// ---- DUTs/ST_COM_SpdCntrl_IMD.TcDUT
TYPE ST_COM_SpdCntrl_IMD :
STRUCT
	StartFormingA		: BOOL;	//Speedcontrol needs the IMD to start froming for A side	
	StartFormingB		: BOOL;	//Speedcontrol needs the IMD to start froming for B side	
	StopForming			: BOOL;					// Speedcontrol needs the IMD to stop forming 
	BlowOffPulseA		: ARRAY[1..4] OF BOOL;	// Blowoff pulses for A side
	BlowOffPulseB		: ARRAY[1..4] OF BOOL;	// Blowoff pulses for B side
	ErrSlotANotFree		: BOOL;					// Current slot for gantry A blow off was not free
	ErrSlotBNotFree		: BOOL;					// Current slot for gantry B blow off was not free
	Modulo				: LREAL;				// Actual modulo position of the belt  
	SpeedInKo			: LREAL;				//Actual Speed that speedcontrol is dictating to the IMD
	PocketA_Blocked		: BOOL;					//Pocket is occupied and gantry is not allowed to blow off
	PocketB_Blocked		: BOOL;					//Pocket is occupied and gantry is not allowed to blow off
	ProdParameters		: St_BlowOffProdPar;	// Needs to be changed to correct format
END_STRUCT
END_TYPE

// ---- DUTs/ST_Record.TcDUT
TYPE ST_Record :
	STRUCT
		nID			: LINT;
		dtTimestamp : DATE_AND_TIME;
		sName		: STRING;
		nSensor1	: LREAL;
	END_STRUCT
END_TYPE

// ---- DUTs/ST_SysPar.TcDUT
TYPE ST_SysPar :
STRUCT
	InMoldDrying					: ST_IMDSysPar;
	ProductHandling					: ST_ProductHandlingSysPar;
END_STRUCT
END_TYPE

// ---- POUs/InMoldDrying/BottomMold/ST_BottomMoldErrors.TcDUT
TYPE ST_BottomMoldErrors :
STRUCT
	VacuumSection						: ARRAY [1..GVL.MaxNrOfVacSectTakeOutUnit] OF BOOL;
	HorizontalCilinder					: ST_CilinderErrors;
	VerticalCilinder					: ST_CilinderErrors;

	Hydraulic							: ST_HydraulicErrors;
	HeatingZone 						: ARRAY [1..6] OF ST_HeatingZoneErrors;
	
	HorizontalAxis						: ST_NcAxis_Errors;
END_STRUCT
END_TYPE

// ---- POUs/InMoldDrying/BottomMold/ST_BottomMoldMachPar.TcDUT
TYPE ST_BottomMoldMachPar :
STRUCT
	EnableNewTakeOut						: BOOL;
	PositionInStop							: REAL;
	//PositionInSlow						: REAL;
	PositionOutStop							: REAL;
	PhysicalOffsetPos						: REAL;
	
	StartVacAtTrPosOffset					: REAL;	// Start vacuum position at postion x of transfer (ofset)			
	StopVacAtBmPosOffset					: REAL; // Stop vacuum at a certain bottommold pos (this is the ofset from the end)
	
	HorizontalCilinder						: ST_CilinderParameters;
	VerticalCilinder						: ST_CilinderParameters;
	
	//BottomMoldVacuumDelay					: TIME := T#22S;
	BottomMoldVacuumClosed					: TIME;
	ClosedVacEnabled						: BOOL;	

	
	VerticalCilinderUpDelay					: TIME := T#1250MS;
	VerticalCilinderTakeOutTime				: TIME := T#1250MS;
	
	
	AxisVelocityManual						: LREAL;
	AxisVelocityInit						: LREAL;
	AxisVelocityAuto						: LREAL;
	AxisPositionRest						: LREAL;
	AxisPositionHome						: LREAL;(* Used when motor is Replaced, write this value as "position bias" in system manager NC-Axis *)

	
	
	//PIDTempZone 							: ARRAY [1..6] OF ST_PIDSettings;
	HeatingZone								: ARRAY [1..6] OF ST_HeatingZone;
	VacuumSection							: ARRAY [1..6] OF FB_MonoValveNoFdbck;
	EnableVacuumSection						: ARRAY [1..6] OF BOOL;	
	
	KickOffCounter							: DINT; // Counts the number of times the bottommold moved in or out.
	GreasingVelocity						: LREAL;
	GreasingPosition						: LREAL;
	
END_STRUCT
END_TYPE

// ---- POUs/InMoldDrying/BottomMold/ST_BottomMoldProdPar.TcDUT
TYPE ST_BottomMoldProdPar :
STRUCT
	par1: REAL;
	
	
END_STRUCT
END_TYPE

// ---- POUs/InMoldDrying/BottomMold/ST_BottomMoldSysPar.TcDUT
TYPE ST_BottomMoldSysPar :
STRUCT
	BottomMoldAxis				: ST_NcAxis_SysPar;
END_STRUCT
END_TYPE

// ---- POUs/InMoldDrying/HydrolicsMain/ST_HydraulicsMainErrors.TcDUT
TYPE ST_HydraulicsMainErrors :
STRUCT
	// Alarms
	OilTemperatureTooHigh				: BOOL;
	OilLevelTooLow						: BOOL;
	Filter100Dirty						: BOOL;
	AuxFilter100Dirty					: BOOL;
	
	// Warnings
	Filter75Dirty						: BOOL;
	AuxFilter75Dirty					: BOOL;
	
	CoolingFanCabinet					: BOOL;
	Hydraulics24VError					: BOOL;
	
	
	// Alarms/Warnings
	HydraulicPump						: ST_MotorSSErrors;
	FilterMotor							: ST_MotorErrors;
	Coolingfan							: ST_MotorErrors;
END_STRUCT
END_TYPE

// ---- POUs/InMoldDrying/HydrolicsMain/ST_HydraulicsMainMachPar.TcDUT
TYPE ST_HydraulicsMainMachPar :
STRUCT
	TempOilCoolingOn			: REAL:= 45;
	TempOilCoolingOff			: REAL:= 30;
	OverTemperature				: REAL:= 50;	
END_STRUCT
END_TYPE

// ---- POUs/InMoldDrying/ProductForming/ST_FormingMoldErrors.TcDUT
TYPE ST_FormingMoldErrors :
STRUCT
	
	Error1: BOOL;

END_STRUCT
END_TYPE

// ---- POUs/InMoldDrying/ProductForming/ST_FormingMoldMachPar.TcDUT
TYPE ST_FormingMoldMachPar :
STRUCT
	VacuumTime							: TIME;
	SecondVacuum						: TIME;
	ThirdVacuum							: TIME := T#300S ;
	VacuumTimeIncr						: TIME; (* Increase vacuum time when pulp tank is switched *)
	BubbleTime							: TIME;
	ClosedTime							: TIME;
	
	StopVacuumAtTrPosOffset				: REAL; // Transfermold endposition minus this ofset is where the forming vacuumvalve is closed.
	StartBlowOffAtTrPosOffset			: REAL; // Transfermold endposition minus this ofset is where the foming mold blowoff is started.
	StopBlowOffAtTrPosOffset			: REAL; // Transfermold endposition minus this ofset is where the forming mold blowoff is stopped.
	


END_STRUCT
END_TYPE

// ---- POUs/InMoldDrying/ProductForming/ST_MachinePondErrors.TcDUT
TYPE ST_MachinePondErrors :
STRUCT
	FeedingPulp							: ST_CilinderErrors;
END_STRUCT
END_TYPE

// ---- POUs/InMoldDrying/ProductForming/ST_MachinePondMachPar.TcDUT
TYPE ST_MachinePondMachPar :
STRUCT
	PositionUpStop						: REAL;
	PositionUpSlow						: REAL;
	PositionDownSlow					: REAL;
	PositionDownStop					: REAL;


	PositionOffsetZero					: REAL;
	PositionOffsetSlowRange				: REAL;
	PositionOffsetAlarm					: REAL;
	
	FeedingPulpTime						: TIME;
	
	BubblingPositionOffset				: REAL;
	
	PositionPhyscialMeasured			: REAL;
	PositionPhysicalMeasuredOld			: REAL;
	PhysicalOffsetPos					: REAL;

	Hydraulic							: ST_HydraulicErrors;
	FeedingPulp							: ST_CilinderParameters;
	Drain								: ST_CilinderParameters;
END_STRUCT
END_TYPE

// ---- POUs/InMoldDrying/ProductForming/ST_ProductFormingErrors.TcDUT
TYPE ST_ProductFormingErrors :
STRUCT
	LowLvlOnBothTanks : BOOL;
	CssHasError: BOOL;
	
	FormingMold					: ST_FormingMoldErrors;
	MachinePond					: ST_MachinePondErrors;
	SprayBar					: ST_SpraybarErrors;
	HydraulicPump				: ST_MotorErrors;
END_STRUCT
END_TYPE

// ---- POUs/InMoldDrying/ProductForming/ST_ProductFormingMachPar.TcDUT
TYPE ST_ProductFormingMachPar :
STRUCT
(*
 (* Forming Mold *)
	MoldVacuum						: FB_MonoValveNoFdbck;							
	MoldBlowOff						: FB_MonoValveNoFdbck;
(* MachinePond *)
	PondHydrolicCilinder			: FB_HydrolicCilinder;
	HydroPump						: FB_HydroPump;
	FeedingPulp						: FB_BiValve2Fdbck;
	Drain							: FB_BiValve2Fdbck;
(* SprayBart *)	
	WireSprayValve					: FB_MonoValveNoFdbck;
	FlashSprayValve					: FB_MonoValveNoFdbck;
	SprayBarMotor					: FB_NCAxis;	
 *)
 
	FormingMold							: ST_FormingMoldMachPar;
	MachinePond							: ST_MachinePondMachPar;
	SprayBar							: ST_SpraybarMachPar;
	
END_STRUCT
END_TYPE

// ---- POUs/InMoldDrying/ProductForming/ST_ProductFormingSysPar.TcDUT
TYPE ST_ProductFormingSysPar :
STRUCT
	SprayBar				: ST_NcAxis_SysPar;
	
END_STRUCT
END_TYPE

// ---- POUs/InMoldDrying/ProductForming/ST_SpraybarErrors.TcDUT
TYPE ST_SpraybarErrors :
STRUCT
	NCAxisError						: ST_NcAxis_Errors;

END_STRUCT
END_TYPE

// ---- POUs/InMoldDrying/ProductForming/ST_SpraybarMachPar.TcDUT
TYPE ST_SpraybarMachPar :
STRUCT
	PositionRestFront					: LREAL;
	PositionRestBack					: LREAL;
	PositionStartFlashFwd				: LREAL;
	PositionStopFlashFwd				: LREAL;
	PositionStartWireFwd				: LREAL;
	PositionStopWireFwd					: LREAL;
	PositionStartFlashBkw				: LREAL;
	PositionStopFlashBkw				: LREAL;
	PositionStartWireBkw				: LREAL;
	PositionStopWireBkw					: LREAL;

	ManualVelocity						: LREAL;
	AutoVelocity						: LREAL;

	PositionActualMeasured				: LREAL; (* ?? *)	
	PositionOffsetZero					: LREAL; (* Zero offset *)

	SprayDelayTime						: TIME;	//Obsolete ("Bateu 20190326")
	SprayDelayTimeOffset				: TIME;	//Spray delay time offset (from 2nd vacuum).
	
	WireSprayInterval					: INT; (* 0 = no spraying *)
	FlashSprayInterval					: INT; (* 0 = no spraying *)
	
	PositionHome						: LREAL;
	
END_STRUCT
END_TYPE

// ---- POUs/InMoldDrying/ST_IMDErrors.TcDUT
TYPE ST_IMDErrors :
STRUCT

	RH_TrMoldIsMovingBoMoldANotInPos	: BOOL; (* RedHot SafetyRule, Transfermold is moving, Bottom Mold A not in position *)
	RH_TrMoldIsMovingBoMoldBNotInPos	: BOOL; (* RedHot SafetyRule, Transfermold is moving, Bottom Mold B not in position *)
	RH_TrMoldIsMovingSprayBNotInPos		: BOOL; (* RedHot SafetyRule, Transfermold is moving, spray bar not in position *)
	RH_SprayBIsMovingTrNotClear			: BOOL;	(* RedHot safetyRule, Spraybar starts moving while transfer is still down on forming*)
	RH_ToMoldAIsMovingBoMoldANotInPos	: BOOL; (* RedHot SafetyRule, Topmold A is moving, Bottom Mold A not in position *)
	RH_ToMoldBIsMovingBoMoldBNotInPos	: BOOL; (* RedHot SafetyRule, Topmold B is moving, Bottom Mold B not in position *)
	RH_BoMoldAIsMovingTrMoldNotInPos	: BOOL; (* RedHot SafetyRule, Bottommold A is moving, Transfermold not in position *)
	RH_BoMoldBIsMovingTrMoldNotInPos	: BOOL; (* RedHot SafetyRule, Bottommold B is moving, Transfermold not in position *)
	RH_BoMoldAIsMovingToMoldANotInPos	: BOOL; (* RedHot SafetyRule, Bottommold A is moving, Topmold A not in position *)
	RH_BoMoldBIsMovingToMoldBNotInPos	: BOOL; (* RedHot SafetyRule, Bottommold B is moving, Topmold B not in position *)
	RH_TaOutHorAIsMovingVertIsNotDown	: BOOL; (* RedHot SafetyRule, Takeout unit Horizontal A is moving, Vertical not in position*)
	RH_TaOutHorBIsMovingVertIsNotDown	: BOOL; (* RedHot SafetyRule, Takeout unit Horizontal A is moving, Vertical not in position*)
	RH_BotMoldAToCoolForTrMDown			: BOOL; (* RedHot SafetyRule, BottomoldA temperature not high enough, and transfer moving down*)
	RH_BotMoldBToCoolForTrMDown			: BOOL; (* RedHot SafetyRule, BottomoldB temperature not high enough, and transfer moving down*)
	
	(* In Auto mode and in Manual Mode. Closing not possible *)
	TempDiffTopBottomTooHigh_SideA		: BOOL; (* Temp Difference Top/Bottom > 20 °C (use average temp)*) 	
	TempDiffTopBottomTooHigh_SideB		: BOOL; (* Temp Difference Top/Bottom > 20 °C (use average temp)*) 	
	
	TempDeviationToHighA				: ARRAY[1..6] OF BOOL;
	TempDeviationToHighB				: ARRAY[1..6] OF BOOL;
	
	TopMoldA							: ST_TopMoldErrors;
	TopMoldB							: ST_TopMoldErrors;
	BottomMoldA							: ST_BottomMoldErrors;
	BottomMoldB							: ST_BottomMoldErrors;
	TransferMold						: ST_TransferMoldErrors;
	ProductForming						: ST_ProductFormingErrors;
	HydraulicMain						: ST_HydraulicsMainErrors;	
END_STRUCT
END_TYPE

// ---- POUs/InMoldDrying/ST_IMDMachPar.TcDUT
TYPE ST_IMDMachPar :
STRUCT
	EnableEamcSideA						: BOOL;
	EnableEamcSideB						: BOOL;
	
	CommisioningMode					: BOOL;	(* Enables movement without RHSR checks.*)
	
	MinTempAlowTransferToBot			: REAL := 175.0;	
	MinimumTransferPosRHSR				: REAL := 950.0;
	MinimumTrDownSprayReleasePosRHSR	: REAL := 750.0;

	
	MinimumTmAPosToAllowBmMove			: REAL := 5.0;		// Offset to Topmold up pos.
	MinimumTmBPosToAllowBmMove			: REAL := 5.0;
	
	MinimumTrUpSprayReleasePosRHSR		: REAL := 300.0;
	SprayBTrCollisionOffset				: REAL := 10.0;
	
	MinimumTrUpSprayReleasePosRHSR2		: REAL := 350.0;
	SprayBTrCollisionOffset2			: REAL := 50.0;
		
	TopMoldA							: ST_TopMoldMachPar;
	TopMoldB							: ST_TopMoldMachPar;
	BottomMoldA							: ST_BottomMoldMachPar;
	BottomMoldB							: ST_BottomMoldMachPar;
	TransferMold						: ST_TransferMoldMachPar;
	ProductForming						: ST_ProductFormingMachPar;
	HydraulicsMain						: ST_HydraulicsMainMachPar;
	
END_STRUCT
END_TYPE

// ---- POUs/InMoldDrying/ST_IMDProdPar.TcDUT
TYPE ST_IMDProdPar :
STRUCT
	TopMoldA				: ST_TopMoldProdPar;
	TopMoldB				: ST_TopMoldProdPar;
	BottomMoldA				: ST_BottomMoldProdPar;
	BottomMoldB				: ST_BottomMoldProdPar;
	TransferMold			: ST_TransferMoldProdPar;
	
END_STRUCT
END_TYPE

// ---- POUs/InMoldDrying/ST_IMDSysPar.TcDUT
TYPE ST_IMDSysPar :
STRUCT
	ProductForming						: ST_ProductFormingSysPar;
	BottomMoldA							: ST_BottomMoldSysPar;
	BottomMoldB							: ST_BottomMoldSysPar;
END_STRUCT
END_TYPE

// ---- POUs/InMoldDrying/TopMold/ST_TopMoldErrors.TcDUT
TYPE ST_TopMoldErrors :
STRUCT
	TmDidNotReachBmPosTimeOut	: BOOL;
	Hydraulic					: ST_HydraulicErrorsAnalog;
	HeatingZone 				: ARRAY [1..6] OF ST_HeatingZoneErrors;
END_STRUCT
END_TYPE

// ---- POUs/InMoldDrying/TopMold/ST_TopMoldMachPar.TcDUT
TYPE ST_TopMoldMachPar :
STRUCT
	EnableClosedBlowOff					: BOOL;
	EnableClosedVacuum					: BOOL;
	BlowOffTimeClosed					: TIME;
	VacuumTimeClosed					: TIME;


// Moving up
	SpeedUpNormal						: REAL;
	SpeedUpSlow							: REAL;
	SpeedUpCreep						: REAL;
	PositionUpStop						: REAL;
	PositionUpSlow						: REAL;
	PositionUpCreep						: REAL;	(*New since speed upgrade*)

// Opening
	SpeedOpening						: REAL;
	//PositionDownOpen					: REAL;	//product par.
	
// Moving down	
	SpeedDownNormal						: REAL;
	SpeedDownSlow						: REAL;
	SpeedDownCreep						: REAL;
	PositionDownSlow					: REAL;
	PositionDownCreep					: REAL;
	//PositionDownStop					: REAL;	// product par.
	
	
// Moving down pressing.
	PressSpeed							: REAL; // Flow at which the pressing is executed.
	PressStop							: REAL; // Pressure at which the pressing stops.

	PositionOffsetZero					: REAL;
	PositionOffsetSlowRange				: REAL;
	PositionOffsetAlarm					: REAL;
	PositionPhyscialMeasured			: REAL;
	PositionPhysicalMeasuredOld			: REAL;
	PhysicalOffsetPos					: REAL;
	
	DryingTime							: TIME;
	BlowOffToTakeOut					: TIME;
	HeatingZone 						: ARRAY [1..6] OF ST_HeatingZone;
END_STRUCT
END_TYPE

// ---- POUs/InMoldDrying/TopMold/ST_TopMoldProdPar.TcDUT
TYPE ST_TopMoldProdPar :
STRUCT

	PositionDownStop			: REAL;
	PositionDownOpen			: REAL;
	
END_STRUCT
END_TYPE

// ---- POUs/InMoldDrying/TransferMold/ST_TransferMoldErrors.TcDUT
TYPE ST_TransferMoldErrors :
STRUCT
	HydraulicCilinder			: ST_HydraulicErrorsAnalog;

	Error1: BOOL;
	Error2: BOOL;

END_STRUCT
END_TYPE

// ---- POUs/InMoldDrying/TransferMold/ST_TransferMoldMachPar.TcDUT
TYPE ST_TransferMoldMachPar :
STRUCT

	PositionUpStop						: REAL;	(* Up *)
	PositionUpSlow						: REAL;	(* Slow up *)
	PositionUpCreep						: REAL;
	
// To Forming	
	PositionDownSlow					: REAL; (* Slow down to forming mold *)
	PositionDownCreep					: REAL;
	UpCreepSpeed						: REAL; (* Transfer Creep speed*)
	UpSlowSpeed							: REAL;	(* Transfer Slow speed*)
	UpNormalSpeed						: REAL; (* Transfer Normal speed*)
	DownSpeed							: REAL; 
	DownSpeedSlow						: REAL;
	DownSpeedCreep						: REAL;
	DownOpenSpeed						: REAL; (* Down open, just above the pond *)

// To bottommold
	PositionTransferSlow				: REAL;	(* Transfer slow *)
	PositionTransferCreep				: REAL;	(* Transfer Creep position*)	
	UpCreepSpeedToBm					: REAL; (* Transfer Creep speed*)
	UpSlowSpeedToBm						: REAL;	(* Transfer Slow speed*)
	UpNormalSpeedToBm					: REAL; (* Transfer Normal speed*)
	DownSpeedToBm						: REAL; 
	DownSpeedSlowToBm					: REAL;
	DownSpeedCreepToBm					: REAL;
	DownOpenSpeedToBm					: REAL; (* Down open, just above the pond *)
	
// To Pause							
	PausePositionUp						: REAL;
	PausePositionUpSlow					: REAL;	// Offset to pause up position 
	PausePositionUpCreep				: REAL;	// Offset to pause up position

// Init speeds
	InitUpCreepSpeed					: REAL; (* Transfer Creep speed*)
	InitUpSlowSpeed						: REAL;	(* Transfer Slow speed*)
	InitUpNormalSpeed					: REAL; (* Transfer Normal speed*)
	InitDownNormalSpeed					: REAL; 
	InitDownSpeedSlow					: REAL;
	InitDownSpeedCreep					: REAL;

// Manual speeds
	ManSpeed							: REAL;
	ManSpeedSlow						: REAL;
	ManSpeedCreep						: REAL;
	
// Misc vars
	PositionStartFormingProcess			: REAL;
	TransferTimeClosed					: TIME;	// Time the transfermold is closed on the bottommold.
	
	PosDownStartVacOffset				: REAL; // Offset voor vacuum valve to open (above forming).
	PosTrStopVacOffset					: REAL; // Offset on the transferposition (above bottomM) for stopping vacuum
	PosTrStartBlowOffOffset				: REAL; // Offset on the transferposition (above bottomM) for opening blow-off
	PosTrStopBlowOffOffset				: REAL; // Offset on the transferposition (above bottomM) for closing blow-off
	
	PositionOffsetZero					: REAL;
	PositionOffsetSlowRange				: REAL;
	PositionOffsetAlarm					: REAL;

	PositionPhyscialMeasured			: REAL;
	PositionPhysicalMeasuredOld			: REAL;
	PhysicalOffsetPos					: REAL;

	
	
	
END_STRUCT
END_TYPE

// ---- POUs/InMoldDrying/TransferMold/ST_TransferMoldProdPar.TcDUT
TYPE ST_TransferMoldProdPar :
STRUCT


	PositionTransferStopA				: REAL;	(* Transfer stop, At Mold B *)
	PositionTransferStopB				: REAL;	(* Transfer stop, At Mold A *)
	PositionTransferOpen				: REAL;	(* Transfer Open, just above the bottom mold *)
	PositionDownStop					: REAL; (* Down stop at forming mold *)
	PositionDownOpen					: REAL; (* Down open, just above the pond *)
	ReleaseBmMovementOffset				: REAL; // Position of the transfermold, that indicates the bottommold is free to move
END_STRUCT
END_TYPE

// ---- POUs/ProductHandling/ST_BlowOffProdPar.TcDUT
TYPE ST_BlowOffProdPar :
STRUCT
	PitchGantry             : DINT;  //Pitch distance between sheets on gantry
	NrOfSheets              : DINT;  //Amount of sheets used on IMD
	NrOfCavities			: DINT;  // The amount of cavities (products) in one sheet.
	Modulo                  : LREAL; //System parameter (5180)
    ModuloOffsetSensorFree		: REAL; //Offset on the modulo to start measuring if the pitch is free for dropping
	ModuloDetectionSensorFree	: REAL;	//How long the sensor needs to be active before alarm/skipping blow off based on modulo length
	SheetSize					: REAL;	//The width of a sheet
END_STRUCT
END_TYPE

// ---- POUs/ProductHandling/ST_GantryMachPar.TcDUT
TYPE ST_GantryMachPar :
STRUCT
	Vert_VelocityManual					: LREAL;
	Vert_VelocityAuto					: LREAL;
	Vert_PositionTransport				: LREAL;
	Vert_PositionHome					: LREAL;(* Used when motor is Replaced, write this value as "position bias" in system manager NC-Axis *)
	Vert_PickUpRestPosOffset			: LREAL; // OffsetPosition in which the gantry waits to pickup product from takeout
	
	Hor_VelocityManual					: LREAL;
	Hor_VelocityAuto					: LREAL;
	Hor_PositionHome					: LREAL;(* Used when motor is Replaced, write this value as "position bias" in system manager NC-Axis *)
	PositionHorizontalPickup			: LREAL;
	PositionHorizontalDropOff			: LREAL;

	EnableVacuumSection					: ARRAY [1..6] OF BOOL;
	
	GantryPickupTime					: TIME := T#500MS;
	
	SheetsProduced						: DINT;	// For OEE, total number of sheets produced by this side (A or B).
	ProductsProduced					: DINT; // For OEE, Total number of products produced
	
END_STRUCT
END_TYPE

// ---- POUs/ProductHandling/ST_GantryProdPar.TcDUT
TYPE ST_GantryProdPar :
STRUCT
	PositionHorizontalPickup			: LREAL;
	PositionHorizontalDropOff			: LREAL;
	PositionVerticalPickup				: LREAL;
	PositionVerticalDropOff				: LREAL;
	
	BlowOffTime							: TIME;
	
END_STRUCT
END_TYPE

// ---- POUs/ProductHandling/ST_GantryErrors.TcDUT
TYPE ST_GantryErrors :
STRUCT
	Collision					: BOOL;
	EndLimitHorFront			: BOOL;
	EndLimitHorBack				: BOOL;
	EndLimitVertUp				: BOOL;
	EndLimitVertDown			: BOOL;
	ProductLost					: ARRAY [1..6] OF BOOL;
	
	VerticalNCAxisError			: ST_NcAxis_Errors;
	HorizontalNCAxisError		: ST_NcAxis_Errors;
END_STRUCT
END_TYPE

// ---- POUs/ProductHandling/ST_GantrySysPar.TcDUT
TYPE ST_GantrySysPar :
STRUCT
	HorizontalAxis				: ST_NcAxis_SysPar;
	VerticalAxis				: ST_NcAxis_SysPar;	
END_STRUCT
END_TYPE

// ---- POUs/ProductHandling/ST_ProductHandlingErrors.TcDUT
TYPE ST_ProductHandlingErrors :
STRUCT
	RH_HorMovingVertNotAtTranspPos_A	: BOOL; (* RedHot SafetyRule, Horizontal is moving when vertical is not at transport position *)
	RH_HorMovingVertNotAtTranspPos_B	: BOOL; (* RedHot SafetyRule, Horizontal is moving when vertical is not at transport position *)
	RH_VertMovingHorNotInPos_A			: BOOL;	(* RedHot SafetyRule, Vertical is moving when horizontal is not at pick or drop position *)
	RH_VertMovingHorNotInPos_B			: BOOL;	(* RedHot SafetyRule, Vertical is moving when horizontal is not at pick or drop position *)

	Gantry_A							: ST_GantryErrors;
	Gantry_B							: ST_GantryErrors;
	
END_STRUCT
END_TYPE

// ---- POUs/ProductHandling/ST_ProductHandlingMachPar.TcDUT
TYPE ST_ProductHandlingMachPar :
STRUCT
	GantryA						: ST_GantryMachPar;
	GantryB						: ST_GantryMachPar;
	CommisioningMode 			: BOOL	:= FALSE;
END_STRUCT
END_TYPE

// ---- POUs/ProductHandling/ST_ProductHandlingProdPar.TcDUT
TYPE ST_ProductHandlingProdPar :
STRUCT
	GantryA						: ST_GantryProdPar;
	GantryB						: ST_GantryProdPar;
	OutfeedConveyor				: ST_OutfeedConveyorProdPar;

END_STRUCT
END_TYPE

// ---- POUs/ProductHandling/ST_ProductHandlingSysPar.TcDUT
TYPE ST_ProductHandlingSysPar :
STRUCT
	GantryA						: ST_GantrySysPar;
	GantryB						: ST_GantrySysPar;
END_STRUCT
END_TYPE

// ---- POUs/Standard/Balluff/ST_BalluffDevice.TcDUT
TYPE ST_BalluffDevice :
STRUCT
	ErrorRegister	: BYTE;
	Temperature	: INT;
	
END_STRUCT
END_TYPE

// ---- POUs/Standard/Balluff/ST_BalluffMagnet.TcDUT
TYPE ST_BalluffMagnet :
STRUCT
	Position	: DINT;
	Speed	: DINT;
	PosMarkerFailure : BYTE;
	CamState1	 : BYTE;
	CamState2	: BYTE;
	CamState3	: BYTE;
	CamState4	 : BYTE;
	PosAboveWorkAreaHighLimit	 : BYTE;
	PosBelowWorkAreaLowLimit	: BYTE;

END_STRUCT
END_TYPE

// ---- POUs/Standard/HeatingZone/PID/ST_PIDSettings.TcDUT
TYPE ST_PIDSettings :
STRUCT
	AutoState		: BOOL;
	SetpointState	: BOOL;
	OutState		: BOOL;	

	//PID_ON			: BOOL;			// PID controller on / off
	IL_ON			: BOOL; 			// Interlock output on 	
	RAUT_OP			: BOOL; 			// Release automatic operation 		
	DEADBAND		: REAL; 		(* Deadband +/- SP-PV *)
	OUT_ROC_UP		: REAL; 		(* Output rate of change up *)
	OUT_ROC_DOWN	: REAL; 		(* Output rate of change down *)
	EU_LLM			: REAL; 		(* Low limit engineerings units SP en PV *)
	EU_HLM			: REAL:= 100.0;	(* High limit engineerings units SP en PV *)
	SP_AUTO			: REAL; 		(* Setpoint Auto *)
	SP_ROC_EXT		: REAL; 		(* Setpoint rate of change *)
	SP_LLM_EXT		: REAL; 		(* Setpoint low limit *)
	SP_HLM_EXT		: REAL:= 100.0;	(* Setpoint high limit *)							
	PV_TMLAG		: REAL; 			// Process value 1ste orde filter (Sec) 	
	SP_MAN			: REAL;
	SP_PID			: REAL;
	fI_InnerWindow	: REAL; 		(*Linear reduction of I component in the innerwindow*)
	INVERTED		: BOOL;		(* (0) PV<SP dan OUT en (1) PV<SP dan OUT *)
	FF_SIGNAL		: REAL;				// Feedforward signal	
	FF_GAIN			: REAL;		(* Feedforward gain	*)
	P				: REAL;		(* P-factor			*)
	I				: REAL; 		(* I-factor (Sec)		*)
	D				: REAL; 		(* D-factor (Sec)		*)
	Dtime			: REAL;		(* Damping time		*)
	TMLAG			: REAL;
	OUT_IL			: REAL; 		(* Output interlock value *)
	OUT_LLM_EXT		: REAL; 			// Output low limit 								
	OUT_HLM_EXT		: REAL:=100.0; 			// Output high limit 	
	OUT_MIN			: REAL; 		(* Output minimum value *)
	OUT_MAX			: REAL:= 100.0;	(* Output maximum value *)
	OUT_MAN			: REAL;		(* Output manual		*)
	OUT_FF			: REAL;		(* Output Feedforward component	*)
	SP_AUTO_TOTAL	: REAL := 185.0;
	LowCutOff		: REAL;
	HighCutOff		: REAL;
	
END_STRUCT
END_TYPE

// ---- POUs/Standard/HeatingZone/ST_HeatingZoneErrors.TcDUT
TYPE ST_HeatingZoneErrors :
STRUCT
	Thermal							: BOOL;
	
	PT100_Loose						: BOOL; (* Alarm 1 -> Main alarm for alarms 2,3, 4 and 5 indicating somethings wrong with pt100*)
	PT100_WireBreak					: BOOL; (* Alarm 2 -> Terminal has detected a wirebreak.*)
	PT100_HasWrongPosition			: BOOL; (* Alarm 3 -> Temperature change detected during startup on PT100 which shouldn't be active.*)
	PT100_NotInserted				: BOOL; (* Alarm 4 -> No Temperature change detected during startup on PT100 while zone is active*)
	PT100_ConnectorNotConnected		: BOOL; (* Connector pt100 not connected: 100 ohm missing / pt100 , open loop.*)
	PT100_TempAboveSetpoint			: BOOL; (* When heating is on, and startup period is over, temperature is higher that 20 degrees above setpoint for a period of 1 minute*)
	PT100_TempBelowSetpoint			: BOOL; (* When heating is on, and startup period is over, temperature is lower that 20 degrees below setpoint for a period of 1 minute*)
	PT100_Heating100OhmTryActivate	: BOOL; (* Happens when the connector measures 100 ohm if this happens, this element may not be enabeled (because of electric failure) *)
	PT100_TemperatureTooHighWarn	: BOOL; (* Temperature too high warning (230 degree) *)
	PT100_TemperatureAboveMaximum	: BOOL;	(* Temperature is above the 250 degree maximum mark.*)
END_STRUCT
END_TYPE

// ---- POUs/Standard/HeatingZone/ST_HeatingZone.TcDUT
TYPE ST_HeatingZone :
STRUCT
	mxEnableZone 			: BOOL;
	mxZoneActive 			: BOOL;
	nrOfSteps				: INT	:= 1;
	LowLimitSP				: REAL  :=130;
	WaitTimeAfterStepReached: TIME := T#30S;
	
	TempErrorRaise			: REAL := 1.0;
	TimeErrorCheckinterval	: TIME := T#15S; 

	
	PWM_Parameters			: ST_CTRL_PWM_OUT_PARAMS;
	PIDTempZone 			: ST_PIDSettings;
	
END_STRUCT
END_TYPE

// ---- POUs/Standard/HydraulicCylinderAnalog/ST_HydraulicCilinderMachParAnalog.TcDUT
TYPE ST_HydraulicCilinderMachParAnalog :
STRUCT
	Hysteresis			: REAL := 2.0;
	MaxRodSidePressure	: REAL := 100.0;
	MaxBotSidePressure	: REAL := 100.0;
END_STRUCT
END_TYPE

// ---- POUs/Standard/HydraulicCylinderAnalog/ST_HydraulicErrorsAnalog.TcDUT
TYPE ST_HydraulicErrorsAnalog:
STRUCT
	//PositionError						: BOOL; (* Out of range *)
	IsMovingWithoutActivation			: BOOL; (* Moving cilinder when no valve is activated *)
	BallufError							: BOOL;

	RodSidePressureTooHigh				: BOOL;	(*Pressure on the Rod side was to high while moving*)
	BotSidePressureTooHigh				: BOOL; (*Pressure on the Bot side was to high while moving*)
	
	SafePositionValveNotReached			: BOOL;
END_STRUCT
END_TYPE

// ---- POUs/Standard/Motor/ST_MotorSSErrors.TcDUT
TYPE ST_MotorSSErrors :
STRUCT	
	SofstarterFailure		: BOOL;
	Maintenance				: BOOL;
END_STRUCT
END_TYPE

// ---- POUs/Standard/HydraulicCilinder/ST_HydraulicCilinderMachPar.TcDUT
TYPE ST_HydraulicCilinderMachPar :
STRUCT
	MainOilPressure : REAL;
	MainFlowPressure: REAL;
	Hysteresis		: REAL := 10.0;
END_STRUCT
END_TYPE

// ---- POUs/Standard/HydraulicCilinder/ST_HydraulicErrors.TcDUT
TYPE ST_HydraulicErrors:
STRUCT
	PositionError						: BOOL; (* Out of range *)
	IsMovingWithoutActivation			: BOOL; (* Moving cilinder when no valve is activated *)
	BallufError							: BOOL;
END_STRUCT
END_TYPE

// ---- POUs/Standard/NC_Axis/ST_NcAxis_Errors.TcDUT
TYPE ST_NcAxis_Errors :
STRUCT
	exDriveStatus: BOOL;
	///~ (OPC:1:available for OPC Clients) 
	exDrivePower: BOOL;
	///~ (OPC:1:available for OPC Clients) 
	exDriveJog: BOOL;
	///~ (OPC:1:available for OPC Clients) 
	exDriveReset: BOOL;
	///~ (OPC:1:available for OPC Clients) 

	exDriveAbsoluut				: BOOL;
	exDriveVelocity				: BOOL;
	exDriveStop					: BOOL;
	exWriteParameter			: BOOL;
	exReadParameter				: BOOL;
	exHome						: BOOL;
	exLagError					: BOOL;	(*Lag error*)
	
END_STRUCT
END_TYPE

// ---- POUs/Standard/Motor/ST_MotorErrors.TcDUT
TYPE ST_MotorErrors :
STRUCT	
	Thermal					: BOOL;
	Maintenance				: BOOL;
END_STRUCT
END_TYPE

// ---- POUs/Standard/NC_Axis/ST_NcAxis_Parameters_XX.TcDUT
TYPE ST_NcAxis_Parameters_XX :
STRUCT
	VelocityAuto		:	LREAL;	(*Automatic speed*)
	VelocityManual		:	LREAL; 	(*manual speed*)
	VelocityInit		:	LREAL;	(*init speed*)
	HomePosition		:	LREAL;	(*Homing position*)
	Acceleration		:	LREAL;  (*Acceleration speed*)
	Deceleration		:	LREAL;  (*Deceleration speed*)
	DecelerationStop	:	LREAL:=1000;	(*Deceleration *)	

END_STRUCT
END_TYPE

// ---- POUs/Standard/NC_Axis/ST_NcAxis_SysPar.TcDUT
TYPE ST_NcAxis_SysPar :
STRUCT
	PositionBias			: LREAL;(* From absolute encoder *)
	IDXGRP				:UDINT := 16#5011;

END_STRUCT
END_TYPE

// ---- POUs/Standard/Valves/ST_CilinderErrors.TcDUT
TYPE ST_CilinderErrors :
STRUCT
	Cilinder					: BOOL;(* Check sensor/cilinder *)
	CilinderSlow_IN				: BOOL;(* Cilinder slow in *)
	CilinderSlow_OUT			: BOOL;(* Cilinder slow out *)
END_STRUCT
END_TYPE

// ---- POUs/Standard/Valves/ST_CilinderParameters.TcDUT
TYPE ST_CilinderParameters :
STRUCT
	T_GuardTimeError				: TIME:=T#500MS;
	T_GuardTimeWarning_IN			: TIME:=T#100MS;
	T_GuardTimeWarning_OUT			: TIME:=T#100MS;
END_STRUCT
END_TYPE

// ---- POUs/ST_Errors.TcDUT
TYPE ST_Errors :
STRUCT
	exEmergency						: ARRAY[1..GVL.MAX_ZONES+1] OF BOOL;  (*Emergecy Stop Active, Index=Zone, 1=Stacker, 2=Zipper, 3=Bundle Buffer track, 4=Vertical denester, 5=Bundle Outfeed // stop buttons.*)
	exEmStopImdFront				: BOOL;
	exEmStopImdBack					: BOOL;
	exEmStopGantryA_Front			: BOOL;
	exEmStopGantryA_Back			: BOOL;
	exEmStopGantryB_Front			: BOOL;
	exEmStopGantryB_Back			: BOOL;
	
	exImdFrontDoorLeft				: BOOL;
	exImdFrontDoorMiddle			: BOOL;
	exImdFrontDoorRight				: BOOL;						
	exImdBackDoorLeft1				: BOOL;
	exImdBackDoorLeft2				: BOOL;
	exImdBackDoorMiddle3			: BOOL;
	exImdBackDoorMiddle4			: BOOL;
	exImdBackDoorRight5				: BOOL;
	exImdBackDoorRight6				: BOOL;

	exGantryA_FrontDoorLeft			: BOOL;
	exGantryA_FrontDoorRight		: BOOL;
	exGantryA_BackDoor				: BOOL;
	exGantryB_FrontDoorLeft			: BOOL;
	exGantryB_FrontDoorRight		: BOOL;
	exGantryB_BackDoor				: BOOL;
	
	MainAirSupplyError				: BOOL;
	
	ex24VoltError1					: BOOL; 
	ex24VoltError2					: BOOL;
	
	exUpsAlarm						: BOOL;
	
	exAtteptedStartWithNoProduct	: BOOL;
	
	InMoldDryingErrors				: ST_IMDErrors;
	ProductHandlingErrors 			: ST_ProductHandlingErrors;
	
	
END_STRUCT
END_TYPE

// ---- GVLs/GVL.TcGVL

VAR_GLOBAL PERSISTENT
	PersMachPar					: ST_MachPar;
	PersSysPar					: ST_SysPar;
END_VAR
VAR_GLOBAL CONSTANT
	MaxNrOfVacSectTakeOutUnit	: INT:= 4;	
	MAX_ZONES					: INT:= 7;
END_VAR

// ---- POUs/MAIN.TcPOU
PROGRAM MAIN
VAR	
	unixTime: UnixTimestamp;
	timestampNanoseconds: ULINT;

	// General variables
	mxReset									: BOOL;
	mxEmergency								: BOOL;
	EmButtons								: BOOL;
	mxAutoMode								: BOOL; (* "1" = Auto, "0" = Manual *)
	mxFirstCycle							: BOOL;
	mxErrorInit								: BOOL;
	mxInitialized							: BOOL;
	SR_AttemptedStartWithNoProductLoaded	: SR;
	
	// Sub objects
	InMoldDrying							: FB_InMoldDrying;
	ProductHandling							: FB_ProductHandling;
	Blink									: FB_Blink;

	// Variables for parameter structs and error structs
	ComSC									: ST_Com_SpeedControl;	// Communication struct for speedcontrol
	MachPar									: ST_MachPar;
	ProductPar								: ST_ProdPar;
	SysPar									: ST_SysPar;
	Errors									: ST_Errors;
	OEEpar									: ST_OEE;
	
	// Variables for/with HMI purposes
{Region "HMI variables"}
	mxHMI_Start								: BOOL;
	mxHMI_Stop								: BOOL;
	mxHMI_Pause								: BOOL;
	mxHMI_Sample							: BOOL;
	mxHMI_Reset								: BOOL;
	mxHMI_StartInit							: BOOL;
	mxHMI_StopInit							: BOOL;
	mxHMI_EnableHeating						: BOOL;

	mxHMI_StartState						: BOOL;
	mxHMI_StopState							: BOOL;
	mxHMI_PauseState						: BOOL;
	mxHMI_SampleState						: BOOL;
	mxHMI_Stopping							: BOOL;
	mxHMI_StartHydraulicsState				: BOOL;
	mxHMI_StopHydraulicsState				: BOOL;
	mxHMI_StartHydraulics					: BOOL;
	mxHMI_StopHydraulics					: BOOL;
	mxHydraulicsReady						: BOOL;
	mxProductLoaded							: BOOL;
	mxMachineInRest							: BOOL;
	
	// Speedcontrol states for hmi
	mrHMI_SpeedControlModulo				: LREAL;
	mxHMI_StartFormingPulse					: BOOL;
	mxHMI_StopFormingPulse					: BOOL;
	mxHMI_SlotANotFree						: BOOL;
	mxHMI_SlotBNotFree						: BOOL;
	mxHMI_IMDHasES							: BOOL;
	mrHMI_MaximumNrOfKickoffs				: REAL;
	mrHMI_ActNrOfKickoffs					: REAL;
	mxHMI_IMDRTO							: BOOL;
	mxHMI_IMDStopped						: BOOL;
	mxHMI_IMDRunning						: BOOL;
	mrHMI_DictatedKoSpeedControl			: LREAL;
	
	
	T_HMIReset								: TON;
	FT_AutoMode								: F_Trig;
	RT_MasterReset							: R_trig;
{End region}
	
	// Triggers for starting and stopping
	RT_Start								: R_TRIG;
	RT_Stop									: R_TRIG;
	RT_StopBySC								: R_TRIG;
	RT_StartBySC							: R_TRIG;
	RT_Pause								: R_TRIG;
	RT_StartInit							: R_TRIG;
	RT_StopInit								: R_TRIG;
	RT_StopOnLowLvl							: R_TRIG;
	RT_StartHydraulics						: R_TRIG;
	RT_StopHydraulics						: R_TRIG;	

	RT_PauseReqGantryA						: R_TRIG;
	RT_PauseReqGantryB						: R_TRIG;
	RT_PauseReqProdHandling					: R_TRIG;
	RT_PauseReqImd							: R_TRIG;
	
	// 24Volt error
	ix24VoltError1							AT %I* : BOOL;
	ix24VoltError2							AT %I* : BOOL;
	SR_24VError1							: SR;
	SR_24VError2							: SR;	
	
	// inputs and ouputs regarding safety 
{Region "Safety variables"}
	ixTwinSafe_SafetyRelay 					AT %I*:ARRAY[1..GVL.MAX_ZONES] OF BOOL; (* couple to zones in Safety programm FB outputs *)
	qxTwinSafe_Reset						AT %Q*: BOOL;
	FbError 								AT %I*: BOOL;
	ComErr 									AT %I*: BOOL;
	OutErr 									AT %I*: BOOL;
	
	(* Operator side/Front *)
	ixResetImdFront							AT %I* : BOOL;
	ixDoorReqImdFront						AT %I* : BOOL;
	qxLightEmStopImdFront					AT %Q* : BOOL;
	qxLightDoorReqImdFront					AT %Q* : BOOL;
	ixEmStopImdFront						AT %I* 	: ARRAY[0..1] OF BOOL; (* couple to the TwinSAFE inputs *)
	(* NON Operator side/Back *)
	ixResetImdBack							AT %I* : BOOL;
	ixDoorReqImdBack						AT %I* : BOOL;
	qxLightEmStopImdBack					AT %Q* : BOOL;
	qxLightDoorReqImdBack					AT %Q* : BOOL;
	ixEmStopImdBack							AT %I* 	: ARRAY[0..1] OF BOOL; (* couple to the TwinSAFE inputs *)

	(* Safety door switches *)
	ixSafetyFrontDoorLeft					AT %I* 	: ARRAY[0..1] OF BOOL; (* couple to the TwinSAFE inputs *)
	ixSafetyFrontDoorMiddle					AT %I* 	: ARRAY[0..1] OF BOOL; (* couple to the TwinSAFE inputs *)
	ixSafetyFrontDoorRight					AT %I* 	: ARRAY[0..1] OF BOOL; (* couple to the TwinSAFE inputs *)
	ixSafetyBackDoorLeft1					AT %I* 	: ARRAY[0..1] OF BOOL; (* couple to the TwinSAFE inputs *)
	ixSafetyBackDoorLeft2					AT %I* 	: ARRAY[0..1] OF BOOL; (* couple to the TwinSAFE inputs *)
	ixSafetyBackDoorMiddle3					AT %I* 	: ARRAY[0..1] OF BOOL; (* couple to the TwinSAFE inputs *)
	ixSafetyBackDoorMiddle4					AT %I* 	: ARRAY[0..1] OF BOOL; (* couple to the TwinSAFE inputs *)
	ixSafetyBackDoorRight5					AT %I* 	: ARRAY[0..1] OF BOOL; (* couple to the TwinSAFE inputs *)
	ixSafetyBackDoorRight6					AT %I* 	: ARRAY[0..1] OF BOOL; (* couple to the TwinSAFE inputs *)

	ixResetGantryA_Front					AT %I* : BOOL;
	ixDoorReqGantryA_Front					AT %I* : BOOL;
	qxLightEmStopGantryA_Front				AT %Q* : BOOL;
	qxLightDoorReqGantryA_Front				AT %Q* : BOOL;
	ixEmStopGantryA_Front					AT %I* 	: ARRAY[0..1] OF BOOL; (* couple to the TwinSAFE inputs *)

	ixResetGantryA_Back						AT %I* : BOOL;
	ixDoorReqGantryA_Back					AT %I* : BOOL;
	qxLightEmStopGantryA_Back				AT %Q* : BOOL;
	qxLightDoorReqGantryA_Back				AT %Q* : BOOL;
	ixEmStopGantryA_Back					AT %I* 	: ARRAY[0..1] OF BOOL; (* couple to the TwinSAFE inputs *)

	ixResetGantryB_Front					AT %I* : BOOL;
	ixDoorReqGantryB_Front					AT %I* : BOOL;
	qxLightEmStopGantryB_Front				AT %Q* : BOOL;
	qxLightDoorReqGantryB_Front				AT %Q* : BOOL;
	ixEmStopGantryB_Front					AT %I* 	: ARRAY[0..1] OF BOOL; (* couple to the TwinSAFE inputs *)

	ixResetGantryB_Back						AT %I* : BOOL;
	ixDoorReqGantryB_Back					AT %I* : BOOL;
	qxLightEmStopGantryB_Back				AT %Q* : BOOL;
	qxLightDoorReqGantryB_Back				AT %Q* : BOOL;
	ixEmStopGantryB_Back					AT %I* 	: ARRAY[0..1] OF BOOL; (* couple to the TwinSAFE inputs *)
	
	ixSafetyGantryA_FrontDoorLeft			AT %I* 	: ARRAY[0..1] OF BOOL; (* couple to the TwinSAFE inputs *)
	ixSafetyGantryA_FrontDoorRight			AT %I* 	: ARRAY[0..1] OF BOOL; (* couple to the TwinSAFE inputs *)
	ixSafetyGantryA_BackDoor				AT %I* 	: ARRAY[0..1] OF BOOL; (* couple to the TwinSAFE inputs *)
	ixSafetyGantryB_FrontDoorLeft			AT %I* 	: ARRAY[0..1] OF BOOL; (* couple to the TwinSAFE inputs *)
	ixSafetyGantryB_FrontDoorRight			AT %I* 	: ARRAY[0..1] OF BOOL; (* couple to the TwinSAFE inputs *)
	ixSafetyGantryB_BackDoor				AT %I* 	: ARRAY[0..1] OF BOOL; (* couple to the TwinSAFE inputs *)
{End Region}
	
	// Emergency stops
	SR_exEmergency							: ARRAY[1..GVL.MAX_ZONES] OF SR; (* Emergency of the zones *)
	SR_EmStopImdFront						: SR;
	SR_EmStopImdBack						: SR;
	SR_EmStopGantryA_Front					: SR;
	SR_EmStopGantryA_Back					: SR;
	SR_EmStopGantryB_Front					: SR;
	SR_EmStopGantryB_Back					: SR;
	
	// Emergency Doors IMD
	SR_SafetyFrontDoorLeft					: SR;
	SR_SafetyFrontDoorMiddle				: SR;
	SR_SafetyFrontDoorRight					: SR;
	SR_SafetyBackDoorLeft1					: SR;
	SR_SafetyBackDoorLeft2					: SR;
	SR_SafetyBackDoorMiddle3				: SR;
	SR_SafetyBackDoorMiddle4				: SR;
	SR_SafetyBackDoorRight5					: SR;
	SR_SafetyBackDoorRight6					: SR;
	DoorRequestImdFront						: GateRequest;
	DoorRequestImdBack						: GateRequest;
	DoorRequestGantryAFront					: GateRequest;
	DoorRequestGantryABack					: GateRequest;
	DoorRequestGantryBFront					: GateRequest;
	DoorRequestGantryBBack					: GateRequest;
	
	// Emergency Doors Gantries
	SR_SafetyGantryA_FrontDoorLeft			: SR;	
	SR_SafetyGantryA_FrontDoorRight			: SR;
	SR_SafetyGantryA_BackDoor				: SR;
	SR_SafetyGantryB_FrontDoorLeft			: SR;	
	SR_SafetyGantryB_FrontDoorRight			: SR;
	SR_SafetyGantryB_BackDoor				: SR;

	// Presistent data
	ChkMachPar								: ST_MachPar;
	CmpMachPar								: DINT;
	ChkSysPar								: ST_SysPar;
	CmpSysPar								: DINT;
	RTRIG_WritePersistent					: R_TRIG;
	FB_WritePersistentData					:  WritePersistentData;
	FB_GetCurTaskIdx						: GETCURTASKINDEX;
	T_WritePersistent						: TON;
	
	// Variables for the ethercat diagnosing.
	iwDevID									AT %I* :UINT;
	iAmsNetID								AT %I* :ARRAY [0..5] OF BYTE;
	iwSlaveCount							AT %I* :UINT;
	iwCfgSlaveCount							AT %I* :UINT;
	iwDevState								AT %I* :UINT;
	EtherCatDiag							:FB_EtherCATDiag;
	AmsNetID								: STRING;
	DeviceID								: INT;
	
	PlcCycleTime     						: REAL := 10.0;
	
	// Variables for O.E.E
	L1										AT %I* : ST_PowerMeasurement;
	L2										AT %I* : ST_PowerMeasurement;
	L3										AT %I* : ST_PowerMeasurement;	
	ActNrOfKickoffs							: REAL;	
	oldSecond								: INT;
	NTGetTime								: NT_GetTime;
	mxPulseCycle							: BOOL; 				(* Pulse 1 cycle on, 1 cycle off *)
	SysTime									: TIMESTRUCT;
	RT_1SecondTrigger						: R_TRIG;
	
	// Outputs for alarm tower.
	qxLightGreen							AT %Q* : BOOL;
	qxLightYellow							AT %Q* : BOOL;
	qxLightRed								AT %Q* : BOOL;
	qxAlarmHorn								AT %Q* : BOOL;
	
	// Variables for the UPS
	ixMainSwitchOFF							AT %I* : BOOL;	
	ixUPS_Alarm								AT %I* : BOOL;
	ixUPS_BatMode							AT %I* : BOOL;
	ixUPS_Charge							AT %I* : BOOL;
	qxPcRemoteOff							AT %Q* : BOOL;
	T_BatteryMode							: TON;
	T_MaintSwitch							: TON;
	SR_UPSAlarm								: SR;
	mxEmDoors								: BOOL;


	mxIMDUnlocked							: BOOL;
	mxProdHandlingUnlocked					: BOOL;
	mxEmptyByStopSC							: BOOL;

	RT_Sample: R_TRIG;
	mxSample: BOOL;
	RT_RestartAfterDoorOpened: R_TRIG;
	FT_Sample: F_TRIG;
	
	mxReset_ByStartInmold			: BOOL;
	mxReset_ByStartProdHandling		: BOOL;
	RT_InMoldDryingBusy				: R_TRIG;
	RT_ProdHandlingBusy				: R_TRIG;
	
	//Main Air supply
	MainAirSupply					: FB_MonoValveNoFdbck;
	MainAirPressureSwitch	AT %I* 	: BOOL;
	SR_MainAirPressureError			: SR;
	
END_VAR

unixTime();
//timestampMilliseconds := unixTime.milliseconds;
//timestampSeconds := unixTime.seconds;
timestampNanoseconds := unixTime.nanoseconds;

// 					Object Calls				//
FB_GetCurTaskIdx();
mxFirstCycle:= _TaskInfo[FB_GetCurTaskIdx.index].FirstCycle;
PlcCycleTime:= UDINT_TO_REAL(_TaskInfo[FB_GetCurTaskIdx.index].CycleTime/10000);
RemanentData();
Blink();
Objects();
HMIState();

// 					R_Trigs.					//
RT_StartHydraulics(CLK:= mxHMI_StartHydraulics);
RT_StopHydraulics(CLK:= mxHMI_StopHydraulics);
RT_Start(CLK:= mxHMI_Start);// OR (ComSC.SpeedControl_IMD.StartForming AND NOT InMoldDrying.mxInPause));
RT_Stop(CLK:= mxHMI_Stop); 
RT_StartBySC(CLK:= ComSC.SpeedControl_IMD.StartFormingA OR ComSC.SpeedControl_IMD.StartFormingB);
RT_StopBySC(CLK:= ComSC.SpeedControl_IMD.StopForming); 
RT_StopOnLowLvl(CLK:= Main.Errors.InMoldDryingErrors.ProductForming.LowLvlOnBothTanks);
RT_Pause(CLK:= mxHMI_Pause);
RT_Sample(CLK:=mxHMI_Sample);
FT_Sample(CLK:=InMoldDrying.mxSample);
RT_StartInit(CLK:= mxHMI_StartInit);
RT_StopInit(CLK:= mxHMI_StopInit);
RT_MasterReset(CLK:= NOT mxAutoMode);
mxInitialized:= InMoldDrying.mxInitialized AND ProductHandling.mxInitialized;
mxMachineInRest := NOT InMoldDrying.mxCycleBusy AND NOT ProductHandling.mxCycleBusy;


// 					Start the Hydraulics		//
IF (RT_StartHydraulics.Q OR (RT_RestartAfterDoorOpened.Q AND InMoldDrying.HydraulicsMain.mxCycleInPause AND mxAutoMode)) AND NOT mxErrorInit THEN
	InMoldDrying.M_StartHydraulics();
END_IF

// 					Stop hydraulics
IF RT_StopHydraulics.Q THEN
	InMoldDrying.M_StopHydraulics();
END_IF

RT_InMoldDryingBusy(CLK:=InMoldDrying.mxCycleBusy);
RT_ProdHandlingBusy(CLK:=ProductHandling.mxCycleBusy);
IF RT_InMoldDryingBusy.Q THEN
	mxReset_ByStartInmold := TRUE;
END_IF
IF RT_ProdHandlingBusy.Q THEN
	mxReset_ByStartProdHandling := TRUE;
END_IF
IF NOT mxEmptyByStopSC THEN
	mxReset_ByStartInmold := FALSE;
	mxReset_ByStartProdHandling := FALSE;	
END_IF

// 					Start machine				//
IF (RT_Start.Q OR (mxEmptyByStopSC AND NOT ComSC.SpeedControl_IMD.StopForming)) AND mxAutoMode AND mxInitialized AND NOT mxErrorInit AND mxProductLoaded AND mxHydraulicsReady AND NOT mxIMDUnlocked AND NOT mxProdHandlingUnlocked THEN  
	InMoldDrying.M_StartCycle(); 
	ProductHandling.M_StartCycle();
	mxHMI_Stopping :=FALSE;
	IF mxReset_ByStartInmold AND mxReset_ByStartProdHandling THEN
		mxEmptyByStopSC := FALSE;
	END_IF
END_IF

//					IMD Pause (stopinpos)		//
IF RT_PauseReqImd.Q THEN
	InMoldDrying.M_StopCycle();	
	mxEmptyByStopSC := FALSE;
END_IF

//					Producthandling Pause (stopinpos)		//
IF RT_PauseReqProdHandling.Q THEN
	ProductHandling.M_StopCycle();	
	mxEmptyByStopSC := FALSE;
END_IF

//					Normal stop					//
IF ((RT_StopOnLowLvl.Q OR RT_Stop.Q OR RT_StopBySC.Q) AND mxAutoMode) THEN  
	InMoldDrying.M_StopCycleEmpty();  
	Producthandling.M_StopCycleEmpty(); 
	mxHMI_Stopping := TRUE;		
	mxEmptyByStopSC := FALSE;
	IF 	RT_StopBySC.Q AND (ProductHandling.mxCycleBusy OR InMoldDrying.mxCycleBusy) THEN
		mxEmptyByStopSC := TRUE;
	END_IF			
END_IF

//					Init machine				//
IF RT_StartInit.Q AND mxAutoMode AND mxProductLoaded AND NOT mxErrorInit AND mxHydraulicsReady THEN 
	InMoldDrying.M_StartInit(); 
	mxEmptyByStopSC := FALSE;
	Producthandling.M_StartInit(); 
END_IF
IF RT_StopInit.Q OR mxErrorInit THEN
	InMoldDrying.M_StopInit();
	ProductHandling.M_StopInit();
	mxEmptyByStopSC := FALSE;
END_IF

//					Stop direct error			//
IF mxErrorInit OR InMoldDrying.mxErrorInit OR ProductHandling.Errors.Gantry_A.Collision OR ProductHandling.Errors.Gantry_B.Collision THEN
	InMoldDrying.M_StopDirect();
	mxEmptyByStopSC := FALSE;
END_IF

IF mxErrorInit OR ProductHandling.mxErrorInit THEN
	ProductHandling.M_StopDirect();
	mxEmptyByStopSC := FALSE;
END_IF



//					Signal light				//
qxLightEmStopImdFront:= qxLightEmStopImdBack:= qxLightEmStopGantryA_Front:= qxLightEmStopGantryA_Back:= qxLightEmStopGantryB_Front:= qxLightEmStopGantryB_Back := 
	Errors.exEmergency[1] OR Errors.exEmergency[2] OR Errors.exEmergency[3] OR Errors.exEmergency[4] OR Errors.exEmergency[5] OR Errors.exEmergency[6] OR Errors.exEmergency[7];
qxLightRed:= HMI.mxError;
qxLightGreen:= mxHMI_StartState := (InMoldDrying.mxCycleBusy OR ProductHandling.mxCycleBusy) AND NOT mxHMI_PauseState;
qxLightYellow:= FALSE;

//					Reseting					//
T_HMIReset(IN:= mxHMI_Reset,PT:=T#1S);
IF T_hmiReset.Q THEN mxHMI_Reset:=FALSE; END_IF

mxReset:= qxTwinSafe_Reset:= mxHMI_Reset OR ixResetImdFront OR ixResetImdBack OR ixResetGantryA_Front OR ixResetGantryA_Back OR ixResetGantryB_Front OR ixResetGantryB_Back;

//					Master reset				//
IF RT_MasterReset.Q THEN
	InMoldDrying.mxResetCycleState := TRUE;
	InMoldDrying.mxResetInitState := TRUE;
	ProductHandling.mxResetCycleState:= TRUE;
	ProductHandling.mxResetInitState:= TRUE;
	mxEmptyByStopSC := FALSE;
END_IF

// 					Sample button				//
IF RT_Sample.Q THEN
	mxSample:= InMoldDrying.mxSample := TRUE;
END_IF; 

IF FT_Sample.Q THEN
	mxSample:=FALSE;
END_IF


// Get AMS net id and device id for ethercat topology
AmsNetID:= F_CreateAmsNetId(iAmsNetID);
DeviceID:= UINT_TO_INT(iwDevID);

// 					Force HMI bits to zero		//
mxHMI_Start := FALSE;
mxHMI_Stop := FALSE;
mxHMI_Pause := FALSE;
mxHMI_Sample:=FALSE;
mxHMI_StartHydraulics := FALSE;
mxHMI_StopHydraulics:=FALSE;

// Shut of PC when on battery mode or when power was switched off:
T_BatteryMode(IN:=ixUPS_BatMode, PT:=T#30S);
T_MaintSwitch(IN:=ixMainSwitchOFF, PT:=T#5S);

// Uncomment when timers are tested.
qxPcRemoteOff := T_BatteryMode.Q OR T_MaintSwitch.Q;

//Main Air Supply
MainAirSupply.M_On();

ACTION Com_SC:
// Current speed (dictated by Speedcontrol)
IF InMoldDrying.ProductForming.CurrentSpeedSingleKO > 0 THEN
	ComSC.IMD_SpeedControl.ActualSpeed := (60000 / InMoldDrying.ProductForming.CurrentSpeedSingleKO);
END_IF

// Current maximum speed (Calculated on bases of own forming).
ComSC.IMD_SpeedControl.MaximumSpeed := InMoldDrying.CalculateMaxKO.MaxKO;


ComSC.IMD_SpeedControl.RTO := mxAutoMode AND mxInitialized AND NOT mxErrorInit AND mxProductLoaded AND mxHydraulicsReady;
ComSC.IMD_SpeedControl.ES := mxEmergency;
ComSC.IMD_SpeedControl.Stopped := NOT InMoldDrying.mxCycleBusy; // AND NOT ProductHandling.mxCycleBusy;
ComSC.IMD_SpeedControl.HMI_Reset := mxHMI_Reset;
END_ACTION

ACTION Error:
(*Emergency Stop Active Zone x,  Index=Zone , 1=Takeout/Gantr A, 2=Imd Left, 3=Imd Middle, 4=Imd Right, 5=Takeout/Gantry B*, 6=Gantry B *)
SR_exEmergency[1](SET1:= NOT ixTwinSafe_SafetyRelay[1], RESET:=ixTwinSafe_SafetyRelay[1] , Q1=>Errors.exEmergency[1] );
SR_exEmergency[2](SET1:= NOT ixTwinSafe_SafetyRelay[2], RESET:=ixTwinSafe_SafetyRelay[2] , Q1=>Errors.exEmergency[2] );
SR_exEmergency[3](SET1:= NOT ixTwinSafe_SafetyRelay[3], RESET:=ixTwinSafe_SafetyRelay[3] , Q1=>Errors.exEmergency[3] );
SR_exEmergency[4](SET1:= NOT ixTwinSafe_SafetyRelay[4], RESET:=ixTwinSafe_SafetyRelay[4] , Q1=>Errors.exEmergency[4] );
SR_exEmergency[5](SET1:= NOT ixTwinSafe_SafetyRelay[5] , RESET:=ixTwinSafe_SafetyRelay[5], Q1=>Errors.exEmergency[5] );
SR_exEmergency[6](SET1:= NOT ixTwinSafe_SafetyRelay[6] , RESET:=ixTwinSafe_SafetyRelay[6], Q1=>Errors.exEmergency[6] );
SR_exEmergency[7](SET1:= NOT ixTwinSafe_SafetyRelay[7] , RESET:=ixTwinSafe_SafetyRelay[7], Q1=>Errors.exEmergency[7] );

(*InMold Drying *)
SR_EmStopImdFront(SET1:= NOT ixEmStopImdFront[0] OR NOT ixEmStopImdFront[1] , RESET:= mxReset, Q1=> Errors.exEmStopImdFront);
SR_EmStopImdBack(SET1:= NOT ixEmStopImdBack[0] OR NOT ixEmStopImdBack[1] , RESET:= mxReset, Q1=> Errors.exEmStopImdBack);

SR_SafetyFrontDoorLeft(SET1:= NOT ixSafetyFrontDoorLeft[0] OR NOT ixSafetyFrontDoorLeft[1] , RESET:= mxReset, Q1=> Errors.exImdFrontDoorLeft);
SR_SafetyFrontDoorMiddle(SET1:= NOT ixSafetyFrontDoorMiddle[0] OR NOT ixSafetyFrontDoorMiddle[1] , RESET:= mxReset, Q1=> Errors.exImdFrontDoorMiddle);
SR_SafetyFrontDoorRight(SET1:= NOT ixSafetyFrontDoorRight[0] OR NOT ixSafetyFrontDoorRight[1] , RESET:= mxReset, Q1=> Errors.exImdFrontDoorRight);
SR_SafetyBackDoorLeft1(SET1:= NOT ixSafetyBackDoorLeft1[0] OR NOT ixSafetyBackDoorLeft1[1] , RESET:= mxReset, Q1=> Errors.exImdBackDoorLeft1);
SR_SafetyBackDoorLeft2(SET1:= NOT ixSafetyBackDoorLeft2[0] OR NOT ixSafetyBackDoorLeft2[1] , RESET:= mxReset, Q1=> Errors.exImdBackDoorLeft2);
SR_SafetyBackDoorMiddle3(SET1:= NOT ixSafetyBackDoorMiddle3[0] OR NOT ixSafetyBackDoorMiddle3[1] , RESET:= mxReset, Q1=> Errors.exImdBackDoorMiddle3);
SR_SafetyBackDoorMiddle4(SET1:= NOT ixSafetyBackDoorMiddle4[0] OR NOT ixSafetyBackDoorMiddle4[1] , RESET:= mxReset, Q1=> Errors.exImdBackDoorMiddle4);
SR_SafetyBackDoorRight5(SET1:= NOT ixSafetyBackDoorRight5[0] OR NOT ixSafetyBackDoorRight5[1] , RESET:= mxReset, Q1=> Errors.exImdBackDoorRight5);
SR_SafetyBackDoorRight6(SET1:= NOT ixSafetyBackDoorRight6[0] OR NOT ixSafetyBackDoorRight6[1] , RESET:= mxReset, Q1=> Errors.exImdBackDoorRight6);

(* Gantry *)
SR_EmStopGantryA_Front(SET1:= NOT ixEmStopGantryA_Front[0] OR NOT ixEmStopGantryA_Front[1] ,RESET:= mxReset, Q1=> Errors.exEmStopGantryA_Front);
SR_EmStopGantryA_Back(SET1:= NOT ixEmStopGantryA_Back[0] OR NOT ixEmStopGantryA_Back[1] ,RESET:= mxReset, Q1=> Errors.exEmStopGantryA_Back);
SR_EmStopGantryB_Front(SET1:= NOT ixEmStopGantryB_Front[0] OR NOT ixEmStopGantryB_Front[1] ,RESET:= mxReset, Q1=> Errors.exEmStopGantryB_Front);
SR_EmStopGantryB_Back(SET1:= NOT ixEmStopGantryB_Back[0] OR NOT ixEmStopGantryB_Back[1] ,RESET:= mxReset, Q1=> Errors.exEmStopGantryB_Back);

SR_SafetyGantryA_FrontDoorLeft(SET1:= NOT ixSafetyGantryA_FrontDoorLeft[0] OR NOT ixSafetyGantryA_FrontDoorLeft[1] , RESET:= mxReset, Q1=> Errors.exGantryA_FrontDoorLeft);
SR_SafetyGantryA_FrontDoorRight(SET1:= NOT ixSafetyGantryA_FrontDoorRight[0] OR NOT ixSafetyGantryA_FrontDoorright[1] , RESET:= mxReset, Q1=> Errors.exGantryA_FrontDoorRight);
SR_SafetyGantryA_BackDoor(SET1:= NOT ixSafetyGantryA_BackDoor[0] OR NOT ixSafetyGantryA_BackDoor[1] , RESET:= mxReset, Q1=> Errors.exGantryA_BackDoor);
SR_SafetyGantryB_FrontDoorLeft(SET1:= NOT ixSafetyGantryB_FrontDoorLeft[0] OR NOT ixSafetyGantryB_FrontDoorLeft[1] , RESET:= mxReset, Q1=> Errors.exGantryB_FrontDoorLeft);
SR_SafetyGantryB_FrontDoorRight(SET1:= NOT ixSafetyGantryB_FrontDoorRight[0] OR NOT ixSafetyGantryB_FrontDoorright[1] , RESET:= mxReset, Q1=> Errors.exGantryB_FrontDoorRight);
SR_SafetyGantryB_BackDoor(SET1:= NOT ixSafetyGantryB_BackDoor[0] OR NOT ixSafetyGantryB_BackDoor[1] , RESET:= mxReset, Q1=> Errors.exGantryB_BackDoor);

(* Main Air Supply *)
SR_MainAirPressureError(SET1 := NOT MainAirPressureSwitch, RESET:= mxReset, Q1=> Errors.MainAirSupplyError);

(*24V error*)
SR_24VError1(Set1:=NOT ix24VoltError1, Reset:=mxReset, Q1=>Errors.ex24VoltError1); 
SR_24VError2(Set1:=NOT ix24VoltError2, Reset:=mxReset, Q1=>Errors.ex24VoltError2); 
SR_UPSAlarm(Set1:=NOT ixUPS_Alarm, Reset:=mxReset, Q1=>Errors.exUpsAlarm);

SR_AttemptedStartWithNoProductLoaded(Set1:=NOT mxProductLoaded AND (RT_Start.Q OR RT_StartInit.Q), Reset:=mxReset, Q1=>Errors.exAtteptedStartWithNoProduct);

EtherCatDiag(
	SlaveCount:=	iwSlaveCount,
	CfgSlaveCount:=	iwCfgSlaveCount,
	DevState:=		iwDevState);

Errors.exEmergency[8]	:=EmButtons := Errors.exEmStopGantryA_Back OR Errors.exEmStopGantryA_Front OR Errors.exEmStopGantryB_Back OR Errors.exEmStopGantryB_Front OR Errors.exEmStopImdBack OR Errors.exEmStopImdFront;

mxEmDoors	:= Errors.exEmergency[1] OR Errors.exEmergency[2] OR Errors.exEmergency[3] OR 
Errors.exEmergency[4] OR Errors.exEmergency[5] OR Errors.exEmergency[6] OR Errors.exEmergency[7]; 	

mxEmergency := mxEmDoors OR EmButtons;

mxErrorInit:= InMoldDrying.mxErrorInit OR ProductHandling.mxErrorInit OR EmButtons OR Errors.MainAirSupplyError OR
				(NOT InMoldDrying.mxInPause AND NOT ProductHandling.mxInPause AND mxEmDoors); // If door is opened without door req, stopdirect (mxErrorInit).
END_ACTION

ACTION HMIState:
//// ***			Starting stopping pause Sample			***	////
mxHMI_StartHydraulicsState := mxHydraulicsReady;
mxHMI_StopHydraulicsState := NOT mxHydraulicsReady;
mxHMI_StartState:= InMoldDrying.mxCycleBusy AND ProductHandling.mxCycleBusy;
mxHMI_PauseState:= InMoldDrying.mxInPause AND ProductHandling.mxInPause;
mxHMI_StopState:= (NOT InMoldDrying.mxCycleBusy AND NOT ProductHandling.mxCycleBusy) OR mxHMI_Stopping;
mxHMI_IMDRunning := NOT mxHMI_PauseState AND (InMoldDrying.mxCycleBusy OR ProductHandling.mxCycleBusy);
mxHMI_SampleState := mxSample;


//// *** 					Speedcontrol					*** ////

// Status for HMI: Speedcontrol commands for IMD
mrHMI_SpeedControlModulo := ComSC.SpeedControl_IMD.Modulo;
mxHMI_StartFormingPulse := ComSC.SpeedControl_IMD.StartFormingA OR ComSC.SpeedControl_IMD.StartFormingB;
mxHMI_StopFormingPulse := ComSC.SpeedControl_IMD.StopForming;
mxHMI_SlotANotFree := ComSc.SpeedControl_IMD.ErrSlotANotFree;
mxHMI_SlotBNotFree := ComSc.SpeedControl_IMD.ErrSlotBNotFree;

// Status for HMI: IMD commands for Speedcontrol
mxHMI_ImdHasES := ComSC.IMD_SpeedControl.ES;
mrHMI_ActNrOfKickoffs := ComSC.IMD_SpeedControl.ActualSpeed;
mrHMI_MaximumNrOfKickoffs := ComSc.IMD_SpeedControl.MaximumSpeed;
mxHMI_IMDRTO := ComSc.IMD_SpeedControl.RTO;
mxHMI_IMDStopped := ComSC.IMD_SpeedControl.Stopped;
mrHMI_DictatedKoSpeedControl := ComSC.SpeedControl_IMD.SpeedInKo;
END_ACTION

ACTION Objects:
HMI();
Error();
SafetyDoors();
Com_SC();
OEE();

InMoldDrying(
	mxReset:= mxReset, 
	mxEmergency:= Errors.exEmergency,//Errors.exEmergency[1] OR Errors.exEmergency[2] OR Errors.exEmergency[3] OR Errors.exEmergency[4] OR Errors.exEmergency[5] OR Errors.exEmStopImdFront OR Errors.exEmStopImdBack,
	mxAutoMode:= mxAutoMode,
	mxStartFormingA:= ComSC.SpeedControl_IMD.StartFormingA,
	mxStartFormingB:= ComSC.SpeedControl_IMD.StartFormingB,
	mxFirstCycle:= mxFirstCycle,
	mxProductPickedUpGantry_A:= ProductHandling.mxProductPickedUpGantry_A,
	mxProductPickedUpGantry_B:= ProductHandling.mxProductPickedUpGantry_B,
	mxEnableHeating:= mxHMI_EnableHeating,
	mxHydraulicsReady=>mxHydraulicsReady,
	mxGantrysNotBusy:= ProductHandling.mxGantrysNotBusy,
	PlcCycleTime:=PlcCycleTime,
	MachParameters:= MachPar.InMoldDrying, 
	ProdParameters:= ProductPar.InMoldDrying, 
	SysParameters:= SysPar.InMoldDrying,
	mxFormingA_Ready => ComSC.IMD_SpeedControl.FormingReadyA,
	mxFormingB_Ready => ComSC.IMD_SpeedControl.FormingReadyB,
	Errors=> Errors.InMoldDryingErrors);

ProductHandling(
	mxReset:= mxReset, 
	mxEmergency:= Errors.exEmergency,//Errors.exEmergency[1] OR Errors.exEmergency[5] OR Errors.exEmergency[6] OR Errors.exEmergency[7] OR Errors.exEmStopImdFront OR Errors.exEmStopImdBack,
	mxAutoMode:= mxAutoMode,
	mxFirstCycle:=mxFirstCycle,
	mxSideA_Enabled:= InMoldDrying.mxSideAEnabled, //MachPar.InMoldDrying.EnableEamcSideA,
	mxSideB_Enabled:= InMoldDrying.mxSideBEnabled, //MachPar.InMoldDrying.EnableEamcSideB,
	mxEamcIsEmpty:= InMoldDrying.mxIsEmpty,
	mxStopBeforeSCstarted := InMoldDrying.mxStopBeforeSCstarted,
	mxProductReadyAtTakeout_A:= InMoldDrying.mxProductReadyAtTakeout_A,
	mxProductReadyAtTakeout_B:= InMoldDrying.mxProductReadyAtTakeout_B,
	mxStopCycleGantryA:=RT_PauseReqGantryA.Q,
	mxStopCycleGantryB:=RT_PauseReqGantryB.Q,
	GantryA_BlowOffPulse:= ComSC.SpeedControl_IMD.BlowOffPulseA,
	GantryB_BlowOffPulse:= ComSC.SpeedControl_IMD.BlowOffPulseB,
	GantryA_BlowOffSucceded	=> ComSC.IMD_SpeedControl.BlowOffProcessedA,
	GantryB_BlowOffSucceded	=> ComSC.IMD_SpeedControl.BlowOffProcessedB,
	GantryA_InPositionAtBelt=> ComSC.IMD_SpeedControl.GantryA_Ready,
	GantryB_InPositionAtBelt=> ComSC.IMD_SpeedControl.GantryB_Ready,
	NrOfSheets := ComSC.SpeedControl_IMD.ProdParameters.NrOfSheets,
	NrOfCavities := COmSC.SpeedControl_IMD.ProdParameters.NrOfCavities,
	MachParameters:= MachPar.ProductHandling, 
	ProdParameters:= ProductPar.ProductHandling,
	SysParameters:= SysPar.ProductHandling,
	Errors=> Errors.ProductHandlingErrors);

MainAirSupply(
	mxReset:= mxReset, 
	mxEmergency:= , 
	mxAutoMode:= TRUE, 
	RHSR_Blocked:= , 
	SlowValveIsInverted:= , 
	mxDisableManualAutoTrigger:= , 
	mxIsOn=> );
END_ACTION

ACTION OEE:
(* Read actual Systemtime *)
mxPulseCycle := NOT mxPulseCycle;
NTGetTime(START:=mxPulseCycle AND NOT NTGetTime.BUSY , TMOUT:=t#100ms,  TIMESTR=>SysTime );

RT_1SecondTrigger(CLK:=WORD_TO_INT(SysTime.wSecond) <> oldSecond);
IF RT_1SecondTrigger.Q THEN
	oldSecond:=WORD_TO_INT(SysTime.wSecond);
END_IF

// Calculate the voltage to normal format (000.00V)
OEEpar.L1_Voltage := DINT_TO_REAL(L1.iwVoltage) / 10000.0;
OEEpar.L2_Voltage := DINT_TO_REAL(L2.iwVoltage) / 10000.0;
OEEpar.L3_Voltage := DINT_TO_REAL(L3.iwVoltage) / 10000.0;

// Calculate the current to normal format (00.00A)
OEEpar.L1_Current := DINT_TO_REAL(L1.iwCurrent) / 1000.0;
OEEpar.L2_Current := DINT_TO_REAL(L2.iwCurrent) / 1000.0;
OEEpar.L3_Current := DINT_TO_REAL(L3.iwCurrent) / 1000.0;

// Calculate the Powerconsumtion 
OEEpar.L1_Watt := OEEpar.L1_Voltage * OEEpar.L1_Current;
OEEpar.L2_Watt := OEEpar.L2_Voltage * OEEpar.L2_Current;
OEEpar.L3_Watt := OEEpar.L3_Voltage * OEEpar.L3_Current;

// Kickoff's A side
IF InMoldDrying.BottommoldA.NrOfKickOffs <> 0 THEN
	OEEpar.KickOffsAside := (60000 / InMoldDrying.BottommoldA.NrOfKickOffs);
ELSE
	OEEpar.KickOffsAside := 0;
END_IF

// Kickoff's B side
IF InMoldDrying.BottommoldB.NrOfKickOffs <> 0 THEN
	OEEpar.KickOffsBside := (60000 / InMoldDrying.BottommoldB.NrOfKickOffs);
ELSE
	OEEpar.KickOffsBside := 0;
END_IF

// Total Kickoff's
OEEpar.KickOffsBothSides := ComSC.IMD_SpeedControl.ActualSpeed;

// IMD Error time:
IF RT_1SecondTrigger.Q AND (InMoldDrying.mxErrorInit OR InMoldDrying.mxErrorStopinPos) THEN
	OEEpar.ImdErrorTime := OEEpar.ImdErrorTime +1;
END_IF

// ProductHandling Error Time:
IF RT_1SecondTrigger.Q AND (ProductHandling.mxErrorInit OR ProductHandling.mxErrorStopinPos) THEN
	OEEpar.ProductHandingErrorTime := OEEpar.ProductHandingErrorTime +1;
END_IF

// Total run time (time that the machine was in automatic production mode)
IF RT_1SecondTrigger.Q AND (mxAutomode AND mxHMI_IMDRunning) THEN
	OEEpar.TotalRunTime := OEEpar.TotalRunTime +1;
END_IF

// Total wait time (time that the machine was ready, with no error, but wasn't running)
IF RT_1SecondTrigger.Q AND (mxAutomode AND NOT mxHMI_IMDRunning AND mxInitialized) THEN
	OEEpar.TotalWaitTime := OEEpar.TotalWaitTime +1;
END_IF

// Down time (time that the machine was unable to operate cause of an error).
// Total wait time (time that the machine was ready, with no error, but wasn't running)
IF RT_1SecondTrigger.Q AND (mxAutomode AND NOT mxHMI_IMDRunning AND (InMoldDrying.mxErrorInit OR InMoldDrying.mxErrorStopinPos OR 
ProductHandling.mxErrorInit OR ProductHandling.mxErrorStopinPos)) THEN
	OEEpar.TotalDownTime := OEEpar.TotalDownTime +1;
END_IF

// Products for A.
OEEpar.ProducedSheetsASide := Main.MachPar.ProductHandling.GantryA.SheetsProduced;			// Number of sheets that the A side has produced
OEEpar.ProducedProductsAside := Main.MachPar.ProductHandling.GantryA.ProductsProduced;			// Number of Products that the A side has produced

// Products for A.
OEEpar.ProducedSheetsBSide := Main.MachPar.ProductHandling.GantryB.SheetsProduced;			// Number of sheets that the B side has produced
OEEpar.ProducedProductsBside := Main.MachPar.ProductHandling.GantryB.ProductsProduced;			// Number of Products that the B side has produced

// Total produced sheets and products.
OEEpar.TotalProducedSheets := Main.MachPar.ProductHandling.GantryA.SheetsProduced + Main.MachPar.ProductHandling.GantryB.SheetsProduced;	
OEEpar.TotalProducedProducts := Main.MachPar.ProductHandling.GantryA.ProductsProduced + Main.MachPar.ProductHandling.GantryB.ProductsProduced;
END_ACTION

ACTION RemanentData:
IF mxFirstCycle THEN
	MachPar:= PersMachPar;
	SysPar:= PersSysPar;
END_IF

CmpMachPar:= MEMCMP(ADR(MachPar), ADR(ChkMachPar),SIZEOF(ChkMachPar));
CmpSysPar:= MEMCMP(ADR(SysPar), ADR(ChkSysPar),SIZEOF(ChkSysPar));

(* Backup every x min. the persistent parameters *)
T_WritePersistent(IN:= NOT T_WritePersistent.Q , PT:=T#5M);

RTrig_WritePersistent(CLK:= (CmpMachPar <> 0) OR (CmpSysPar <> 0));

IF RTRIG_WritePersistent.Q THEN
	PersMachPar:= MachPar;
	PersSysPar:= SysPar;
	FB_WritePersistentData(NETID:='', PORT:=851, START:=TRUE, TMOUT:=T#1S );	
ELSE
	FB_WritePersistentData(NETID:='', PORT:=851, START:=FALSE, TMOUT:=T#1S );
END_IF

ChkMachPar:= MachPar;
ChkSysPar:= SysPar;
END_ACTION

ACTION SafetyDoors:
{Region "In mold dryer doors"} 
// In mold dryer 
DoorRequestImdFront(
	GateClosed:= NOT Errors.exImdFrontDoorLeft AND NOT Errors.exImdFrontDoorMiddle AND NOT Errors.exImdFrontDoorRight, 
	SafeState:= InMoldDrying.mxInPause AND ProductHandling.mxInPause, 
	Request_Open:= ixDoorReqImdFront, 
	Reset:=mxReset, 
	TimeOutSafeState:= T#10S, 
	Lock=> , 
	GateRequest_Light=> qxLightDoorReqImdFront, 
	ResetButton_Light=> );

DoorRequestImdBack(
	GateClosed:= NOT Errors.exImdBackDoorLeft1 AND NOT Errors.exImdBackDoorLeft2 AND NOT Errors.exImdBackDoorMiddle3 AND NOT Errors.exImdBackDoorMiddle4 
	AND NOT Errors.exImdBackDoorRight5 AND NOT errors.exImdBackDoorRight6, 
	SafeState:= InMoldDrying.mxInPause AND ProductHandling.mxInPause, 
	Request_Open:= ixDoorReqImdBack, 
	Reset:=mxReset, 
	TimeOutSafeState:= T#10S, 
	Lock=> , 
	GateRequest_Light=> qxLightDoorReqImdBack, 
	ResetButton_Light=> );
{End Region}
	
{Region "Gantries"}
// Gantry A Front
DoorRequestGantryAFront(
	GateClosed:= NOT Errors.exGantryA_FrontDoorLeft AND NOT Errors.exGantryA_FrontDoorRight, 
	SafeState:= InMoldDrying.mxInPause AND ProductHandling.mxInPause,  
	Request_Open:= ixDoorReqGantryA_Front, 
	Reset:=mxReset, 
	TimeOutSafeState:= T#10S, 
	Lock=> , 
	GateRequest_Light=> qxLightDoorReqGantryA_Front, 
	ResetButton_Light=> );

DoorRequestGantryABack(
	GateClosed:= NOT Errors.exGantryA_BackDoor, 
	SafeState:= InMoldDrying.mxInPause AND ProductHandling.mxInPause,  
	Request_Open:= ixDoorReqGantryA_Back, 
	Reset:=mxReset, 
	TimeOutSafeState:= T#10S, 
	Lock=> , 
	GateRequest_Light=> qxLightDoorReqGantryA_Back, 
	ResetButton_Light=> );

DoorRequestGantryBFront(
	GateClosed:= NOT Errors.exGantryB_FrontDoorLeft AND NOT Errors.exGantryB_FrontDoorRight, 
	SafeState:= InMoldDrying.mxInPause AND ProductHandling.mxInPause, 
	Request_Open:= ixDoorReqGantryB_Front, 
	Reset:=mxReset, 
	TimeOutSafeState:= T#10S, 
	Lock=> , 
	GateRequest_Light=> qxLightDoorReqGantryB_Front, 
	ResetButton_Light=> );
	
DoorRequestGantryBBack(
	GateClosed:= NOT Errors.exGantryB_BackDoor, 
	SafeState:= InMoldDrying.mxInPause AND ProductHandling.mxInPause, 
	Request_Open:= ixDoorReqGantryB_Back, 
	Reset:=mxReset, 
	TimeOutSafeState:= T#10S, 
	Lock=> , 
	GateRequest_Light=> qxLightDoorReqGantryB_Back, 
	ResetButton_Light=> );
{End Region}

// Collect al lockstates.
mxIMDUnlocked := NOT DoorRequestImdFront.Lock OR NOT DoorRequestImdBack.Lock;
mxProdHandlingUnlocked := NOT DoorRequestGantryABack.Lock OR NOT DoorRequestGantryAFront.Lock OR NOT DoorRequestGantryBBack.Lock OR NOT DoorRequestGantryBFront.Lock;
RT_RestartAfterDoorOpened(CLK:=NOT mxIMDUnlocked AND NOT mxProdHandlingUnlocked AND mxReset);


// Handle the requests
RT_PauseReqImd(ClK:=(ixDoorReqImdFront OR ixDoorReqImdBack OR ixDoorReqGantryA_Front OR ixDoorReqGantryB_Front OR InMoldDrying.mxErrorStopinPos) AND mxAutoMode);
//RT_PauseReqGantryA(CLK:=ixDoorReqImdFront OR ixDoorReqImdBack OR ixDoorReqGantryA_Front OR ixDoorReqGantryA_Back);
//RT_PauseReqGantryB(CLK:=ixDoorReqImdFront OR ixDoorReqImdBack OR ixDoorReqGantryB_Front OR ixDoorReqGantryB_Back);
RT_PauseReqProdHandling(CLK:=(ixDoorReqImdFront OR ixDoorReqImdBack OR ixDoorReqGantryB_Front OR ixDoorReqGantryB_Back OR InMoldDrying.mxErrorStopinPos)AND mxAutoMode);
END_ACTION

END_PROGRAM

// ---- POUs/Standard/UnixTimestamp.TcPOU
FUNCTION_BLOCK UnixTimestamp
VAR_OUTPUT
	nanoseconds: ULINT;
END_VAR

VAR
    localSystemTime : FB_LocalSystemTime := ( bEnable := TRUE, dwCycle := 1 );
    getTimeZoneInformation : FB_GetTimeZoneInformation;
    timeZoneInformation : ST_TimeZoneInformation;
    specificLocalTimeToFileTime : FB_TzSpecificLocalTimeToFileTime;
    fileTime: T_FILETIME;
    onZerothSecondLastCycle : BOOL;
END_VAR

// Get local system time
localSystemTime();

// On the zeroth second of each minutesync timezone information
IF (timeZoneInformation.standardName = '' OR (localSystemTime.systemTime.wSecond = 0 AND NOT onZerothSecondLastCycle)) THEN
    getTimeZoneInformation(sNetID := '', bExecute := TRUE, tzInfo => timeZoneInformation);
END_IF;

// Convert local system time to unix timestamps
specificLocalTimeToFileTime(in := Tc2_Utilities.SYSTEMTIME_TO_FILETIME(localSystemTime.systemTime), tzInfo := timeZoneInformation, out => fileTime);
nanoseconds := (SHL(DWORD_TO_ULINT(fileTime.dwHighDateTime), 32) + DWORD_TO_ULINT(fileTime.dwLowDateTime));

onZerothSecondLastCycle := localSystemTime.systemTime.wSecond = 0;

END_FUNCTION_BLOCK

// ---- POUs/InMoldDrying/FB_InMoldDrying.TcPOU
FUNCTION_BLOCK FB_InMoldDrying
(* Objects 
	EAMC
		-TopMold_A, TopMold_B:			
			-HydrolicCilinder:
				-ValveUp
				-ValveDown
				-ValveSlow
			-ValveRelief
			-ValveBlowOff
			-ValveVacuum
		
		-BottomMold_A, BottomMold_B:
			-HydrolicCilinder:
				-ValveUp
				-ValveDown
				-ValveSlow
			-ValveBlowOff
			-ValveVacuum

		-TransferMold
			-HydrolicCilinder:
				-ValveUp
				-ValveDown
				-ValveSlow
			-ValveBlowOff
			-ValveVacuum

		-ProductForming
			-MachinePond
				-HydrolicCilinder:
					-ValveUp
					-ValveDown
					-ValveSlow
			-SprayBar
				-ValveWire
				-ValveBeard
			-FormingMold
				-ValveVacuum
				-ValveBlowOff
		-HydrolicsMain:
			-HydroPump
			-Rebotech
*)
VAR CONSTANT
	sCycleStateTextDef: ARRAY[0..100]  OF STRING :=	
		['State 0: Wait for Start',
		'State 1: Wait for product forming ready',
		'State 2: Wait for transfermold down at forming position',
		'State 3: Wait for productforming time closed',
		'State 4: Moving transfermold up',
		'State 5: spare',
		'State 6: Move bottommold A or B in',
		'State 7: Move transfermold up',
		'State 8: Move bottommold A or B Out',
		'State 9: Move topmold A or B down, await product forming ready',
		'State 10: Wait for transfermold down at forming position',
		'State 11: Move tranfermold up with product',
		'State 12: Await transfer and topmold A or B up to Release bottommold A/ B movement',
		'State 13: Spare',
		'State 14: Spare',
		'State 15: [Emptying] Move topmold A Or B up',
		'State 16: [Emptying] Move bottommold A or B in ',
		'State 17: [Emptying] Move bottommold A or B out',
		'State 18: [Emptying] Waiting on machine to empty',
		'State 19: [Pause] Waiting on subparts to pause',
		'State 20: [Paused]',
		'State 21: [Paused]',
		'State 22: [Emptying] Machine is empty, awaiting producthandling',
		'State 23: [Direct stop]'];
	
	tCycleStateTimeouts: ARRAY[0..10] OF TIME := 
		[T#10S,T#10S,T#10S,T#10S,T#10S,T#10S,T#10S,T#10S,T#10S,T#10S,
		T#10S];

	sInitStateTextDef: ARRAY[0..10] OF STRING :=
		['State 0: Wait for Start',
		'State 1',
		'State 2: Init transfermold and machinepond',
		'State 3: Init top mold A',
		'State 4: Init Bottom mold A',
		'State 5: Init Top mold B',
		'State 6: Init Bottom mold B',
		'State 7: Set initalised bits and stop pump',
		'State 8',
		'State 9',
		'State 10: Stop init state'];

	tInitStateTimeouts: ARRAY[0..10] OF TIME := 
		[T#10S,T#10S,T#10S,T#10S,T#10S,T#10S,T#10S,T#10S,T#10S,T#10S
		,T#10S];
END_VAR

VAR_INPUT
	mxResetCycleState				: BOOL;
	mxResetInitState				: BOOL;
	mxForceInit						: BOOL; (*Reset Calibration Flag*)
	mxReset							: BOOL;	(*Reset Error*)
	mxEmergency						: ARRAY [1..Max_Zones+1] OF BOOL; // 1=TakeOutA, 2=Aside, 3=mid, 4=Bside, 5=TakeoutB, 6= GantryB, 7=GantryA, 8=All EM stop.
	mxAutoMode						: BOOL; (* TRUE = Automode *)
	mxFirstCycle					: BOOL;
	mxEnableHeating					: BOOL;
	
	mxStart							: BOOL;
	mxStop							: BOOL;
	mxPause							: BOOL;
	
	mxtest							: BOOL;
	
	mxPauseReqZone1					: BOOL;
	mxPauseReqZone2					: BOOL;
	mxPauseReqZone3					: BOOL;
	mxPauseReqZone4					: BOOL;
	mxPauseReqZone5					: BOOL;
	mxProductPickedUpGantry_A		: BOOL;
	mxProductPickedUpGantry_B		: BOOL;	
	mxGantrysNotBusy				: BOOL;
	PlcCycleTime					: REAL;
END_VAR
VAR_IN_OUT
	MachParameters					: ST_IMDMachPar;
	ProdParameters					: ST_IMDProdPar;
	SysParameters					: ST_IMDSysPar;
END_VAR
VAR_OUTPUT
(*Errors*)
	Errors							: ST_IMDErrors;
	mxErrorInit						: BOOL;		(* Error, stop immediately. Initialisation neccesary *)
	mxErrorStopinPos				: BOOL;		(* Error, stop in position. Only reset neccesary *)

(* State vars *)
	mxCycleBusy						: BOOL;
	mxInitBusy						: BOOL;

(* Signals *)
	mxProductReadyAtTakeout_A		: BOOL;
	mxProductReadyAtTakeout_B		: BOOL;	
	mxIsEmpty						: BOOL;
(* Vars *)
	mxInitialized					: BOOL;

	mxHydraulicsReady				: BOOL;
END_VAR
VAR
(* State vars *)
	miCycleState					: INT :=0;
	miCycleOldstate					: INT :=0;
	mxCycleTransitionState			: BOOL := FALSE;
	sCycleStateText					: STRING;
	exCycleTimeOut					: BOOL;		(* Timeout for the whole programcycle *)
	CycleTimeout					: TON;
	CycleTimeOutUpFlank				: R_TRIG;
	mxCycleTimeoutEnable			: BOOL;
	CycleTime						: REAL;
	mxCycleHasError					: BOOL;
	miStopState						: INT;
	mxStartCycle					: BOOL;
	mxStopCycle						: BOOL;
	mxStopCycleEmpty				: BOOL;
	mxStopDirect					: BOOL;
	
	miInitState						: INT	:=0;
	miInitOldstate					: INT	:=0;
	mxInitTransitionState			: BOOL	:= FALSE;
	sInitStateText					: STRING;
	exInitTimeOut					: BOOL;		(* Timeout for the whole programcycle *)
	InitTimeout						: TON;
	InitTimeOutUpFlank				: R_TRIG;
	mxInitTimeoutEnable				: BOOL;
	InitTime						: REAL;
	mxInitHasError					: BOOL;
	mxStartInit						: BOOL;
	mxStopInit						: BOOL;
	
(* Objects *)
	TopMoldA		 				: FB_TopMold;
	TopMoldB		 				: FB_TopMold;
	BottomMoldA						: FB_BottomMold;
	BottomMoldB						: FB_BottomMold;
	TransferMold					: FB_TransferMold;
	ProductForming					: FB_ProductForming;
	HydraulicsMain					: FB_HydraulicsMain;

(* Vars *)	
	mxStartTransferToBottomMold		: BOOL;	(* Signal to transfer mold *)


	
	FT_EnableASide					: F_TRIG;
	FT_EnableBSide					: F_TRig;
	
	mxSideAEnabled: BOOL;
	mxSideBEnabled: BOOL;
	
	SR_TrMoldIsMovingBoMoldANotInPos	: SR; (* RedHot SafetyRule, Transfermold is moving, Bottom Mold A not in position *)
	SR_TrMoldIsMovingBoMoldBNotInPos	: SR; (* RedHot SafetyRule, Transfermold is moving, Bottom Mold B not in position *)
	SR_TrMoldIsMovingSprayBNotInPos		: SR; (* RedHot SafetyRule, Transfermold is moving, spray bar not in position *)
	SR_ToMoldAIsMovingBoMoldANotInPos	: SR; (* RedHot SafetyRule, Topmold A is moving, Bottom Mold A not in position *)
	SR_ToMoldBIsMovingBoMoldBNotInPos	: SR; (* RedHot SafetyRule, Topmold B is moving, Bottom Mold B not in position *)
	SR_BoMoldAIsMovingTrMoldNotInPos	: SR; (* RedHot SafetyRule, Bottommold A is moving, Transfermold not in position *)
	SR_BoMoldBIsMovingTrMoldNotInPos	: SR; (* RedHot SafetyRule, Bottommold B is moving, Transfermold not in position *)
	SR_BoMoldAIsMovingToMoldANotInPos	: SR; (* RedHot SafetyRule, Bottommold A is moving, Topmold A not in position *)
	SR_BoMoldBIsMovingToMoldBNotInPos	: SR; (* RedHot SafetyRule, Bottommold B is moving, Topmold B not in position *)
	SR_TaOutHorAIsMovingVertIsNotDown	: SR; (* RedHot SafetyRule, Takeout unit A Horizontal is moving, Vertical not in position*)
	SR_TaOutHorBIsMovingVertIsNotDown	: SR; (* RedHot SafetyRule, Takeout unit A Horizontal is moving, Vertical not in position*)
	RT_ErrorInit						: R_TRIG;
	mxCommisioningMode					: BOOL;
	T_StopCommisioningMode				: TON;
	mxSafetyRulesEnabled				: BOOL;
	mxBSideReady						: BOOL;
	mxAsideReady						: BOOL;
	
	//VacuumTakeout					: ARRAY [1..6] OF FB_MonoValveNoFdbck;	(* IMD-V *)		
	SR_TempDeviationToHighA				: ARRAY[1..6] OF SR;
	SR_TempDeviationToHighB				: ARRAY[1..6] OF SR;
	RT_DryingTimeA: R_TRIG;
	T_AlmTimeCounterA: TON;
	RT_DryingTimeB: R_TRIG;
	T_AlmTimeCounterB: TON;
	ASideNotWarm: BOOL;
	BSideNotWarm: BOOL;
	SR_BotMoldAToCoolForTrMDown: SR;
	SR_BotMoldBToCoolForTrMDown: SR;
	RT_ProcessTimeA: R_TRIG;
	T_AlmProcessTimeCounterA: TON;
	RT_ProcessTimeB: R_TRIG;
	T_AlmProcessTimeCounterB: TON;
	RT_Pause: R_TRIG;
	
	mxInPause : BOOL;
	ProductDryingAtSideA: BOOL;
	ProductDryingAtSideB: BOOL;
	ContinueWithA: BOOL;
	ContinueWithB: BOOL;
	ProductOnTopMoldA: BOOL;
	ProductOnTopMoldB: BOOL;
	T_TransferReleasedBottom: TON;
	T_TopReleasedBottom: TON;
	mxTest3: BOOL;
	mxTest1: BOOL;
	mxTest2: BOOL;
	TransferLateTime: TIME;
	TopLateTime: TIME;
	RT_ReleaseDifference: R_TRIG;
	RT_ChooseSide: R_TRIG;
	mxEmptying: BOOL;
	LastProductWasA: BOOL;
END_VAR

VAR_TEMP
	RT_PauseReqZone5: R_TRIG;
END_VAR

RT_ErrorInit(CLK:= mxErrorInit AND mxCycleBusy);
IF RT_ErrorInit.Q THEN
	mxStopDirect:= TRUE;
END_IF

FT_EnableASide(CLK:= MachParameters.EnableEamcSideA);
FT_EnableBSide(CLK:= MachParameters.EnableEamcSideB);

// IF Bside is not enabeld, and enable of aside is taken away, set A side again automaticaly
IF NOT MachParameters.EnableEamcSideB AND FT_EnableASide.Q AND NOT MachParameters.CommisioningMode THEN
	MachParameters.EnableEamcSideA :=TRUE;
END_IF

// IF Aside is not enabeld, and enable of Bside is taken away, set B side again automaticaly
IF NOT MachParameters.EnableEamcSideA AND FT_EnableBSide.Q AND NOT MachParameters.CommisioningMode THEN
	MachParameters.EnableEamcSideB := TRUE;
END_IF

// Automaticaly log out off commisioning mode after 2hours.
T_StopCommisioningMode(IN:=MachParameters.CommisioningMode, PT:=T#120M);
IF T_StopCommisioningMode.Q THEN
	MachParameters.CommisioningMode := FALSE;
END_IF

(* Actions *)
Error();
ErrorsTemperature();
Init();
Cycle();
Objects();

ACTION Cycle:
(*StateChange (Transition)  Signalgeneration*)
mxCycleTransitionState:=(miCycleState<>miCycleOldstate);
(*State text*)
sCycleStateText:=sCycleStateTextDef[miCycleState];
(*Timeout Watchdog for Statemachine*)
mxCycleTimeoutEnable:=NOT (miCycleState=0) AND NOT mxReset;

CycleTimeout(IN:=mxCycleTimeoutEnable, PT:=tCycleStateTimeouts[miCycleState] );
CycleTimeOutUpFlank(CLK:=CycleTimeout.Q );
miCycleOldstate:=miCycleState;

(*Set Errorbit when Raising edge of Timeout has been detected*)
IF CycleTimeOutUpFlank.Q THEN
	exCycleTimeOut:=TRUE; 			(* 1 Timeout for the whole programcycle *)
END_IF

(*Function to reset the Statemachine*)
IF mxResetCycleState THEN
	mxPause := FALSE;
	mxResetCycleState:= FALSE;
	miCycleState:=0;
	miCycleOldstate:=miCycleState;
	mxCycleTransitionState:=FALSE;

	TopMoldA.mxResetCycleState:= TRUE;
	TopMoldB.mxResetCycleState:= TRUE;
	BottomMoldA.mxResetCycleState:= TRUE;
	BottomMoldB.mxResetCycleState:= TRUE;
	TransferMold.mxResetCycleState:= TRUE;
	ProductForming.mxResetCycleState:= TRUE;
	
	mxInitialized := FALSE;
	mxStartCycle:= FALSE;
	mxStopCycle:= FALSE;
	mxStopCycleEmpty := FALSE;
	mxStopDirect:= FALSE;
	mxASideReady := FALSE;	// Used to determine which side needs attention
	mxBSideReady := FALSE;
	
	T_AlmProcessTimeCounterA.IN:=FALSE;
	T_AlmProcessTimeCounterB.IN:=FALSE;
	T_AlmTimeCounterA.IN := FALSE;
	T_AlmTimeCounterB.IN := FALSE;
	
	ProductDryingAtSideA	  := FALSE;
	ProductDryingAtSideB	  := FALSE;
	
	miStopState:= 0;
END_IF

// Code to unpause when in pause mode.
IF mxCycleBusy AND mxStartCycle THEN
	mxStartCycle:=FALSE;
	IF NOT TopMoldA.mxCycleBusy THEN TopMoldA.M_StartCycle(); END_IF
	IF NOT TopMoldB.mxCycleBusy THEN TopMoldB.M_StartCycle(); END_IF
	IF NOT TransferMold.mxCycleBusy THEN TransferMold.M_StartCycle(); END_IF
	IF NOT BottomMoldA.mxCycleBusy THEN	BottomMoldA.M_StartCycle(); END_IF
	IF NOT BottomMoldB.mxCycleBusy THEN	BottomMoldB.M_StartCycle(); END_IF
	IF NOT ProductForming.mxCycleBusy THEN ProductForming.M_StartCycle(); END_IF
END_IF

(*Definition State has Error*)
mxCycleHasError:=FALSE;

// Only switch sides when machine stands still.
IF NOT mxCycleBusy THEN 
	mxSideAEnabled:= MachParameters.EnableEamcSideA;
	mxSideBEnabled:= MachParameters.EnableEamcSideB;
END_IF



{region "Code to determine: Continue with A /B"}
RT_ChooseSide(CLK:=(miCycleState = 4) OR (miCycleState = 10));

	 IF RT_ChooseSide.Q THEN			// <- Needs to b a R_TRIG	
		IF mxSideAEnabled AND NOT mxSideBEnabled THEN		// Only A enabled
			ContinueWithA := TRUE;
			ContinueWithB := False;
		ELSIF NOT mxSideAEnabled AND mxSideBEnabled THEN 	// Only B enabled
			ContinueWithA := FALSE;
			ContinueWithB := True;
		ELSIF mxSideAEnabled AND mxSideBEnabled THEN		// A AND B enabled
			IF ContinueWithA then							// when busy with A, new carton will be B
				ContinueWithA := FALSE;
				ContinueWithB := TRUE;
			ELSIF ContinueWithB THEN						// When Busy with B, New carton will be A
				ContinueWithA := TRUE;
				ContinueWithB := False;
			END_IF
		END_IF
	END_IF
{endregion}

{region "Determine which signaled for release first."}
	T_TransferReleasedBottom(IN:=, PT:=T#600S);
	T_TopReleasedBottom(IN:=, PT:=T#600S);
	RT_ReleaseDifference(CLK:=(*(NOT (miCycleState = 12)) OR *) NOT mxTest3 , Q=> );

	IF mxTest3 OR miCycleState = 12 THEN //Step 12
		IF TransferMold.sgTrReleaseBmMoveIn OR mxTest1 THEN
			T_TransferReleasedBottom.IN:=TRUE;
		END_IF
		
		IF TopMoldA.SgTmIsUp OR TopMoldB.SgTmIsUp OR mxTest2 THEN
			T_TopReleasedBottom.IN:=TRUE;		
		END_IF
	END_IF
	
	IF RT_ReleaseDifference.Q THEN
		TransferLateTime:=T#0MS;
		TopLateTime:=T#0MS;
		IF T_TransferReleasedBottom.ET > T_TopReleasedBottom.ET THEN
			TransferLateTime := T_TransferReleasedBottom.ET;
		ELSIF T_TopReleasedBottom.ET > T_TransferReleasedBottom.ET THEN
			TopLateTime := T_TopReleasedBottom.ET;
		END_IF	

		T_TransferReleasedBottom.IN:=FALSE;	
		T_TopReleasedBottom.IN:=FALSE;
	END_IF	

{endregion}

{region "Overname uitleg"}	
		(*
		// >>>	Transfer moves down
		// * Forming stops vacuum pos
		// * Transfer start vacuum pos
		// * Closed timer
		// * Blowoff forming mold aan pos
		// * Blowoff forming mold uit pos
		*)
{endregion}

(*Cycle State's*)
CASE miCycleState OF
	0:	// Wait for start 
		IF mxStartCycle THEN
			mxStartCycle:= FALSE;
			miStopState:= 0;
			mxIsEmpty:= FALSE;
			mxEmptying:=FALSE;
			
			//HydraulicsMain.HydraulicPump.M_Start();
			
			IF mxSideAEnabled AND mxSideBEnabled THEN
				ContinueWithB := TRUE;
				ContinueWithA := FALSE;
			END_IF
			
			TransferMold.M_StartCycle();
			ProductForming.M_StartCycle();
			
			IF mxSideAEnabled THEN 
				TopMoldA.M_StartCycle(); 
				BottomMoldA.M_StartCycle();
			END_IF
			IF mxSideBEnabled THEN 
				TopMoldB.M_StartCycle(); 
				BottomMoldB.M_StartCycle();
			END_IF
			
			miCycleState:= 1;
		END_IF
		
	1:	// Wait for product forming ready
		IF mxStopDirect THEN
			mxStopDirect:= FALSE;
			miCycleState:=23;
		ELSIF mxStopCycle THEN
			mxStopCycle:= FALSE;
			miStopState:= miCycleState;
			miCycleState:= 19;
		ELSIF ProductForming.SgTransferToDownForming THEN	// Signal the transfer to move down
			ProductForming.SgTransferToDownForming :=FALSE;
			TransferMold.sgMoveDownToFormingPos:= TRUE;
			miCycleState:= 2;	
		END_IF
		
	2:  // Wait for transfermold is down at forming pos
		IF mxStopDirect THEN
			mxStopDirect:= FALSE;
			miCycleState:=23;
		ELSIF mxStopCycle THEN
			mxStopCycle:= FALSE;
			miStopState:= miCycleState;
			miCycleState:= 19;
		ELSIF TransferMold.sgTrAtFormingPos THEN	
			TransferMold.sgTrAtFormingPos := FALSE;
			ProductForming.sgTransferIsDown:= TRUE;		// ProductForming.TransferAtStopVacuumForming
			miCycleState:= 3;
		END_IF
		
	3: // Wait for productforming time closed and then move transfer up
		IF mxStopDirect THEN
			mxStopDirect:= FALSE;
			miCycleState:=23;
		ELSIF mxStopCycle THEN
			mxStopCycle:= FALSE;
			miStopState:= miCycleState;
			miCycleState:= 19;
		ELSIF ProductForming.sgTransferToMoveUp THEN	// ClosedDelayTimeElapsed
			ProductForming.sgTransferToMoveUp := FALSE;
			TransferMold.sgMoveUp:= TRUE;
			miCycleState:= 4;
		END_IF
	
	4:	// Move Transfermold up and at certain point make a new porduct (only if emty machine is not active).
		IF TransferMold.mxStartProductForming THEN 
			TransferMold.mxStartProductForming:= FALSE;
			ProductForming.mxStartCycle:= TRUE;
		END_IF
	
		//mxEmptying := mxStopCycleEmpty;
		
		// These bits indicate weather it is the first run for a certain side.
		ProductOnTopMoldA := FALSE;
		ProductOnTopMoldB := FALSE;
		
		// These bits indicate if a side is empty
		ProductDryingAtSideA	  := FALSE;
		ProductDryingAtSideB	  := FALSE;
		
		IF mxStopDirect THEN
			mxStopDirect:= FALSE;
			miCycleState:=23;
		ELSIF mxStopCycle THEN
			mxStopCycle:= FALSE;
			miStopState:= miCycleState;
			miCycleState:= 19;
		ELSIF TransferMold.sgTrReleaseBmMoveIn AND ContinueWithA THEN
			TransferMold.sgTrReleaseBmMoveIn:= FALSE;
			BottomMoldA.sgMoveIn:= TRUE;
			BottomMoldA.mxProductOnTopMold:= ProductOnTopMoldA;	// Skip step 5 (move top mold up, because at a fresh start,
			miCycleState := 6;									// topmold is allready up. Just continue with the bottommold in movement.
		ELSIF TransferMold.sgTrReleaseBmMoveIn AND ContinueWithB THEN
			TransferMold.sgTrReleaseBmMoveIn:= FALSE;
			BottomMoldB.mxProductOnTopMold:= ProductOnTopMoldB;
			BottomMoldB.sgMoveIn:= TRUE;
			miCycleState := 6;
		END_IF										
		
		//\\//\\//\\//\\/\\//\\//\\//\\//\\/\\//\\//\\//\\//\\/\\//\\//\\//\\//\\/\\//\\//\\//\\//\\/\\//\\//\\ Main program loop			
	5:	// Obsolete Step.
	
	6:	// Move bottom mold A / B in		
		IF mxStopDirect THEN
			mxStopDirect:= FALSE;	
			miCycleState:=23;
		ELSIF mxStopCycle THEN
			mxStopCycle:= FALSE;
			miStopState:= miCycleState;
			miCycleState:= 19;
		ELSIF BottomMoldA.SgBottomIsIn AND ContinueWithA THEN
			BottomMoldA.SgBottomIsIn := FALSE; 
			TransferMold.sgMoveToTransferPosA:= TRUE;
			miCycleState:= 7;
		ELSIF BottomMoldB.SgBottomIsIn AND ContinueWithB THEN
			BottomMoldB.SgBottomIsIn := FALSE; 
			TransferMold.sgMoveToTransferPosB:= TRUE;
			miCycleState:= 7;
		END_IF

	7:	// Move Transfer mold up
		IF mxStopDirect THEN
			mxStopDirect:= FALSE;	
			miCycleState:=23;
		ELSIF mxStopCycle THEN
			mxStopCycle:= FALSE;
			miStopState:= miCycleState;
			miCycleState:= 19;
		ELSIF Transfermold.sgTransferIsUpMoveOut AND ContinueWithA THEN
			Transfermold.sgTransferIsUpMoveOut := FALSE; 
			TransferMold.sgMoveToTransferPosA:= FALSE;
			BottomMoldA.sgMoveOut:= TRUE;
			miCycleState:= 8;
		ELSIF Transfermold.sgTransferIsUpMoveOut AND ContinueWithB THEN
			Transfermold.sgTransferIsUpMoveOut := FALSE;
			TransferMold.sgMoveToTransferPosB:= FALSE; 
			BottomMoldB.sgMoveOut:= TRUE;
			miCycleState:= 8;
		END_IF
		
	8:	// Move bottom Mold A / B Out
		IF mxStopDirect THEN
			mxStopDirect:= FALSE;
			miCycleState:=23;
		ELSIF mxStopCycle THEN
			mxStopCycle:= FALSE;
			miStopState:= miCycleState;
			miCycleState:= 19;
		ELSIF BottomMoldA.SgBottomIsOut AND ContinueWithA THEN
			BottomMoldA.SgBottomIsOut := FALSE; 
			TopMoldA.sgMoveDown:= TRUE;	
			TransferMold.sgBottomMoldAIsOut := TRUE;		
			miCycleState:= 9;
		ELSIF BottomMoldB.SgBottomIsOut AND ContinueWithB THEN
			BottomMoldB.SgBottomIsOut := FALSE; 
			TopMoldB.sgMoveDown:= TRUE;	
			TransferMold.sgBottomMoldBIsOut := TRUE;		
			miCycleState:= 9;		
		END_IF

	9:	// Move Topmold A / B down, Wait for productForming ready
		IF mxStopDirect THEN
			mxStopDirect:= FALSE;
			miCycleState:=23;
		ELSIF mxStopCycle THEN
			mxStopCycle:= FALSE;
			miStopState:= miCycleState;
			miCycleState:= 19;
		ELSIF (ProductForming.SgTransferToDownForming OR mxEmptying) AND ContinueWithA THEN	
			ProductForming.SgTransferToDownForming:=FALSE; 
			ProductDryingAtSideA := TRUE;
			
			IF mxEmptying THEN
				IF mxSideAEnabled AND mxSideBEnabled THEN
					ContinueWithA := NOT ContinueWithA;
					ContinueWithB := NOT ContinueWithB;
				END_IF
				miCycleState:= 15;
			ELSE
				TransferMold.sgMoveDownToFormingPos:= TRUE;
				miCycleState:= 10;
			END_IF
		ELSIF (ProductForming.SgTransferToDownForming OR mxEmptying) AND ContinueWithB THEN	
			ProductForming.SgTransferToDownForming:=FALSE; 
			ProductDryingAtSideB := True;
			
			IF mxEmptying THEN
				IF mxSideAEnabled AND mxSideBEnabled THEN
					ContinueWithA := NOT ContinueWithA;
					ContinueWithB := NOT ContinueWithB;
				END_IF
				miCycleState:= 15;
			ELSE
				TransferMold.sgMoveDownToFormingPos:= TRUE;
				miCycleState:= 10;
			END_IF				
		END_IF																									
			
	10: // Wait for transfermold is down at forming pos !! Meanwhile, at top of cycle, new continue with A/B is set.
		IF mxStopDirect THEN
			mxStopDirect:= FALSE;
			miCycleState:=23;
		ELSIF mxStopCycle THEN
			mxStopCycle:= FALSE;
			miStopState:= miCycleState;
			miCycleState:= 19;
		ELSIF TransferMold.sgTrAtFormingPos THEN		// No selection is side is done cause its irrelavant here.
			Transfermold.sgTrAtFormingPos := FALSE;
			ProductForming.sgTransferIsDown:= TRUE;
			miCycleState:= 11;
		END_IF

	11: //Wait for productforming after blowOff is on
		IF mxStopDirect THEN
			mxStopDirect:= FALSE;
			miCycleState:=23;
		ELSIF mxStopCycle THEN
			mxStopCycle:= FALSE;
			miStopState:= miCycleState;
			miCycleState:= 19;
		ELSIF ProductForming.sgTransferToMoveUp THEN	// ClosedDelayTimeElapsed
			ProductForming.sgTransferToMoveUp := FALSE;
			TransferMold.sgMoveUp:= TRUE;
			miCycleState:= 12;
		END_IF

	12:	// Move Transfermold up 
		IF TransferMold.mxStartProductForming AND NOT mxStopCycleEmpty THEN 
			TransferMold.mxStartProductForming:= FALSE;
			ProductForming.mxStartCycle:= TRUE;
		END_IF
		
		// Set a bit to show the machine is emptying. This ensures that the transfer loses its last product on the bottommold.
		mxEmptying:=mxStopCycleEmpty;
	
		IF mxStopDirect THEN
			mxStopDirect:= FALSE;
			miCycleState:=23;
		ELSIF mxStopCycle THEN
			mxStopCycle:= FALSE;
			miStopState:= miCycleState;
			miCycleState:= 19;
		ELSIF TransferMold.sgTrReleaseBmMoveIn AND (TopmoldA.SgTmIsUp OR NOT ProductDryingAtSideA) AND ContinueWithA THEN		// A side = next
			TransferMold.sgTrReleaseBmMoveIn:= FALSE;		
			BottomMoldA.sgMoveIn:= TRUE;
			ProductOnTopMoldA := TRUE; 										// Next time this step is executed, the topmold will indicate it has a product
			BottomMoldA.mxProductOnTopMold:= ProductDryingAtSideA;
			miCycleState:= 6;	
		ELSIF TransferMold.sgTrReleaseBmMoveIn AND (TopMoldB.SgTmIsUp OR NOT ProductDryingAtSideB) AND ContinueWithB THEN 		// B Side = next
			TransferMold.sgTrReleaseBmMoveIn:= FALSE;		
			BottomMoldB.sgMoveIn:= TRUE;
			ProductOnTopMoldB := TRUE; 										// Next time this step is executed, the topmold will indicate it has a product
			BottomMoldB.mxProductOnTopMold:= ProductDryingAtSideB;//ProductOnTopMoldB;
			miCycleState:= 6;	
		END_IF

		//\\//\\//\\//\\/\\//\\//\\//\\//\\/\\//\\//\\//\\//\\/\\//\\//\\//\\//\\/\\//\\//\\//\\//\\/\\//\\//\\ Normal production loop -> 6
	13: // Obsolete Step
		miCycleState:=16;
		
	14: // Obsolete Step
		miCycleState:=15;
		
	15:	// Move topmold A / B up 
		IF mxStopDirect THEN
			mxStopDirect:= FALSE;
			miCycleState:=23;
		ELSIF mxStopCycle THEN
			mxStopCycle:= FALSE;
			miStopState:= miCycleState;
			miCycleState:= 19;
		ELSIF TopMoldA.SgTmIsUp AND ContinueWithA THEN
			BottomMoldA.sgMoveIn:= TRUE;
			BottomMoldA.mxProductOnTopMold:= TRUE;
			miCycleState:= 16;
		ELSIF TopMoldB.SgTmIsUp AND ContinueWithB THEN
			BottomMoldB.sgMoveIn:= TRUE;
			BottomMoldB.mxProductOnTopMold:= TRUE;
			miCycleState:= 16;
		END_IF
		
	16: // Move bottomMold in to fill takeoutunit with last product on this side
		IF mxStopDirect THEN
			mxStopDirect:= FALSE;
			miCycleState:=23;
		ELSIF mxStopCycle THEN
			mxStopCycle:= FALSE;
			miStopState:= miCycleState;
			miCycleState:= 19;
		ELSIF BottomMoldA.SgBottomIsIn AND ContinueWithA THEN
			BottomMoldA.SgBottomIsIn := FALSE; 
			BottomMoldA.sgMoveOut:= TRUE;	
			miCycleState:= 17;
		ELSIF BottomMoldB.SgBottomIsIn AND ContinueWithB THEN
			BottomMoldB.SgBottomIsIn := FALSE; 
			BottomMoldB.sgMoveOut:= TRUE;	
			miCycleState:= 17;
		END_IF 
		
	17: // Move bottommold out to the gantries, and wait for last product on this side to be picked up
		IF mxStopDirect THEN
			mxStopDirect:= FALSE;
			miCycleState:=23;
		ELSIF mxStopCycle THEN
			mxStopCycle:= FALSE;
			miStopState:= miCycleState;
			miCycleState:= 19;
		ELSIF BottomMoldA.SgBottomIsOut AND ContinueWithA THEN
			BottomMoldA.SgBottomIsOut := FALSE;
			TopMoldA.mxMoveUp:= TRUE;
			ContinueWithA := FALSE;
			ContinueWithB := TRUE;
			ProductDryingAtSideA := FALSE;
			
			LastProductWasA := TRUE;
			
			IF NOT ProductDryingAtSideA AND NOT ProductDryingAtSideB THEN
				miCycleState:=18;
			ELSE	
				miCycleState:= 15;
			END_IF
		ELSIF BottomMoldB.SgBottomIsOut AND ContinueWithB THEN
			BottomMoldB.SgBottomIsOut := FALSE;
			TopMoldB.mxMoveUp:= TRUE;
			ContinueWithA := TRUE;
			ContinueWithB := FALSE;
			ProductDryingAtSideB := FALSE;
			
			LastProductWasA := FALSE;
			
			IF NOT ProductDryingAtSideA AND NOT ProductDryingAtSideB THEN
				miCycleState:=18;
			ELSE	
				miCycleState:= 15;
			END_IF
		END_IF 

	18:	// Machine is empty, Wait until Gantry picked up Product A and B 
		IF mxStopDirect THEN
			mxStopDirect:= FALSE;
			miCycleState:=23;
		ELSIF mxStopCycle THEN
			mxStopCycle:= FALSE;
			miStopState:= miCycleState;
			miCycleState:= 19;
		ELSIF (LastProductWasA AND BottommoldA.mxHorCilIsIn AND BottomMoldA.mxGantryPickedUpProduct) OR
				(NOT LastProductWasA AND BottommoldB.mxHorCilIsIn AND BottomMoldB.mxGantryPickedUpProduct) THEN 	
			mxIsEmpty := TRUE;
			mxEmptying := FALSE;
			mxStopCycleEmpty := FALSE;
	
			ProductOnTopMoldA := FALSE;
			ProductOnTopMoldB := FALSE;
			
			miStopState:= miCycleState;
			miCycleState:= 21;
		END_IF
	
	19: // stopping sub objects.
		IF TopMoldA.mxCycleBusy THEN TopMoldA.M_StopCycle(); END_IF
		IF TopMoldB.mxCycleBusy THEN TopMoldB.M_StopCycle(); END_IF
		IF TransferMold.mxCycleBusy THEN TransferMold.M_StopCycle(); END_IF
		IF BottomMoldA.mxCycleBusy THEN	BottomMoldA.M_StopCycle(); END_IF
		IF BottomMoldB.mxCycleBusy THEN	BottomMoldB.M_StopCycle(); END_IF
		IF ProductForming.mxCycleBusy THEN ProductForming.M_StopCycle(); END_IF
		IF HydraulicsMain.mxCycleBusy THEN HydraulicsMain.M_StopCycle(); END_IF
		
		miCycleState := 20;
		
	20: // Pause / Stop sub parts.
		IF mxStopDirect THEN
			mxStopDirect:= FALSE;
			miCycleState:=23;
		ELSIF mxStartCycle OR mxtest THEN
			mxStartCycle:= FALSE;
			TopMoldA.M_StartCycle();
			TopMoldB.M_StartCycle();
			TransferMold.M_StartCycle();
			BottomMoldA.M_StartCycle();
			BottomMoldB.M_StartCycle();
			ProductForming.M_StartCycle();

			miCycleState:= miStopState;
		END_IF;
		
	21: // Stop Cycle 
		mxStopCycle:= FALSE;

		IF TopMoldA.mxCycleBusy THEN TopMoldA.M_EmptyMachine(); END_IF
		IF TopMoldB.mxCycleBusy THEN TopMoldB.M_EmptyMachine(); END_IF
		IF TransferMold.mxCycleBusy THEN TransferMold.M_EmptyMachine(); END_IF
		IF BottomMoldA.mxCycleBusy THEN	BottomMoldA.M_EmptyMachine(); END_IF
		IF BottomMoldB.mxCycleBusy THEN	BottomMoldB.M_EmptyMachine(); END_IF
		IF ProductForming.mxCycleBusy THEN ProductForming.M_EmptyMachine(); END_IF

		IF TopMoldA.mxCycleBusy THEN TopMoldA.M_StopCycle(); END_IF
		IF TopMoldB.mxCycleBusy THEN TopMoldB.M_StopCycle(); END_IF
		IF TransferMold.mxCycleBusy THEN TransferMold.M_StopCycle(); END_IF
		IF BottomMoldA.mxCycleBusy THEN	BottomMoldA.M_StopCycle(); END_IF
		IF BottomMoldB.mxCycleBusy THEN	BottomMoldB.M_StopCycle(); END_IF
		IF ProductForming.mxCycleBusy THEN ProductForming.M_StopCycle(); END_IF

		miCycleState:= 22;

	22: // Stop cycle 
		IF mxStopDirect THEN
			mxStopDirect:= FALSE;
			
			miCycleState:=23;
		ELSIF NOT TopMoldA.mxCycleBusy AND NOT TopMoldB.mxCycleBusy AND NOT TransferMold.mxCycleBusy AND NOT BottomMoldA.mxCycleBusy
			AND NOT BottomMoldB.mxCycleBusy AND NOT ProductForming.mxCycleBusy THEN

			BottomMoldA.mxEmptyMachine:= FALSE;
			BottomMoldB.mxEmptyMachine:= FALSE;
			TransferMold.mxStartProductForming := FALSE;			
			miCycleState:= 0;
		END_IF
	
	23: // Stop Direct 
		mxStartCycle:= FALSE;
		mxStopCycle:= FALSE;
		mxStopDirect:= FALSE;
		miStopState:= 0;
		mxInitialized:= FALSE;
		mxStopCycleEmpty := FALSE;
		mxEmptying := FALSE;
		ProductOnTopMoldA := FALSE;
		ProductOnTopMoldB := FALSE;
		
		T_AlmProcessTimeCounterA.IN:=FALSE;
		T_AlmProcessTimeCounterB.IN:=FALSE;
		T_AlmTimeCounterA.IN := FALSE;
		T_AlmTimeCounterB.IN := FALSE;
		
		ProductDryingAtSideA	  := FALSE;
		ProductDryingAtSideB	  := FALSE;
		
		IF HydraulicsMain.mxCycleBusy THEN HydraulicsMain.m_StopDirect(); END_IF
		IF TopMoldA.mxCycleBusy THEN TopMoldA.M_StopDirect(); END_IF
		IF TopMoldB.mxCycleBusy THEN TopMoldB.M_StopDirect(); END_IF
		IF TransferMold.mxCycleBusy THEN TransferMold.M_StopDirect(); END_IF
		IF BottomMoldA.mxCycleBusy THEN	BottomMoldA.M_StopDirect(); END_IF
		IF BottomMoldB.mxCycleBusy THEN	BottomMoldB.M_StopDirect(); END_IF
		IF ProductForming.mxCycleBusy THEN ProductForming.M_StopDirect(); END_IF

		miCycleState:= 0;
END_CASE

mxCycleBusy:= miCycleState<>0;
END_ACTION

ACTION Error:

(********** RED HOT SAFETY RULES ************)
mxSafetyRulesEnabled := ((mxInitialized AND mxAutoMode) OR (NOT mxAutomode)) AND NOT MachParameters.CommisioningMode;

	(* Transfer Mold Up or Down 	Bottom Drying Molds are In or Out / Spray bar is at one of the rest positions *)	
	SR_TrMoldIsMovingBoMoldANotInPos(SET1:=mxSafetyRulesEnabled AND  (TransferMold.mxCilIsMovingIn OR TransferMold.mxCilIsMovingOut) AND 
	(NOT BottomMoldA.mxCilIsOut AND NOT BottomMoldA.mxCilIsIn) AND (TransferMold.ActualPosition < 950) , RESET:= mxReset, Q1=> Errors.RH_TrMoldIsMovingBoMoldANotInPos);
	
	SR_TrMoldIsMovingBoMoldBNotInPos(SET1:= mxSafetyRulesEnabled AND (TransferMold.mxCilIsMovingIn OR TransferMold.mxCilIsMovingOut) AND
	(NOT BottomMoldB.mxCilIsOut AND NOT BottomMoldB.mxCilIsIn) AND (TransferMold.ActualPosition < 950), RESET:= mxReset, Q1=> Errors.RH_TrMoldIsMovingBoMoldBNotInPos);

	SR_TrMoldIsMovingSprayBNotInPos(SET1:= mxSafetyRulesEnabled AND (TransferMold.mxCilIsMovingOut AND NOT ProductForming.mxSprayBarAtRestPos) AND NOT (BottomMoldA.mxCilIsIn OR BottomMoldB.mxCilIsIn),
	RESET:= mxReset, Q1=> Errors.RH_TrMoldIsMovingSprayBNotInPos);
	
	(* Top Drying Mold Down 	Corresponding Bottom Drying Mold Out *)
	SR_ToMoldAIsMovingBoMoldANotInPos(SET1:= mxSafetyRulesEnabled AND TopMoldA.mxCilIsMovingOut AND NOT BottomMoldA.mxCilIsOut, //NOT BottomMoldA.mxCilIsIn, 
		RESET:= mxReset, Q1=> Errors.RH_ToMoldAIsMovingBoMoldANotInPos);
	SR_ToMoldBIsMovingBoMoldBNotInPos(SET1:= mxSafetyRulesEnabled AND TopMoldB.mxCilIsMovingOut AND NOT BottomMoldB.mxCilIsOut, //NOT BottomMoldB.mxCilIsIn, 
		RESET:= mxReset, Q1=> Errors.RH_ToMoldBIsMovingBoMoldBNotInPos);
	
	(* Bottom Drying Mold In	Corresponding Top Drying Mold Up and Transfer Mold is Up *)
	SR_BoMoldAIsMovingToMoldANotInPos(SET1:= mxSafetyRulesEnabled AND BottomMoldA.mxCilIsMovingIn AND NOT TopMoldA.mxCilIsIn, 
		RESET:= mxReset, Q1=> Errors.RH_BoMoldAIsMovingToMoldANotInPos);
	SR_BoMoldAIsMovingTrMoldNotInPos(SET1:= mxSafetyRulesEnabled AND BottomMoldA.mxCilIsMovingIn AND NOT TransferMold.mxCilIsIn, 
		RESET:= mxReset, Q1=> Errors.RH_BoMoldAIsMovingTrMoldNotInPos);
	SR_BoMoldBIsMovingToMoldBNotInPos(SET1:= mxSafetyRulesEnabled AND BottomMoldB.mxCilIsMovingIn AND NOT TopMoldB.mxCilIsIn, 
		RESET:= mxReset, Q1=> Errors.RH_BoMoldBIsMovingToMoldBNotInPos);
	SR_BoMoldBIsMovingTrMoldNotInPos(SET1:= mxSafetyRulesEnabled AND BottomMoldB.mxCilIsMovingIn AND NOT TransferMold.mxCilIsIn, 
		RESET:= mxReset, Q1=> Errors.RH_BoMoldBIsMovingTrMoldNotInPos);
	
	(* Table Horizontal In	Corresponding Table Vertical is down *)	
	SR_TaOutHorAIsMovingVertIsNotDown(SET1:= mxSafetyRulesEnabled AND (NOT BottomMoldA.mxHorCilIsIn AND NOT BottomMoldA.mxVertCilIsOut), // in is down
		RESET:= mxReset, Q1=> Errors.RH_TaOutHorAIsMovingVertIsNotDown);
	SR_TaOutHorBIsMovingVertIsNotDown(SET1:= mxSafetyRulesEnabled AND (NOT BottomMoldB.mxHorCilIsIn AND NOT BottomMoldB.mxVertCilIsOut), // in is down
		RESET:= mxReset, Q1=> Errors.RH_TaOutHorBIsMovingVertIsNotDown);

// OR BottomMoldA.mxErrorStopinPos OR BottomMoldB.mxErrorStopinPos 
(**********************************************************************************************************)
mxErrorStopinPos:= TopMoldA.mxErrorStopinPos OR TopMoldB.mxErrorStopinPos OR BottomMoldA.mxErrorStopinPos OR BottomMoldB.mxErrorStopinPos 
	OR TransferMold.mxErrorStopinPos OR ProductForming.mxErrorStopinPos OR HydraulicsMain.mxErrorStopinPos;	
	
mxErrorInit:= TopMoldA.mxErrorInit OR TopMoldB.mxErrorInit Or BottomMoldA.mxErrorInit Or BottomMoldB.mxErrorInit
	OR TransferMold.mxErrorInit OR ProductForming.mxErrorInit OR HydraulicsMain.mxErrorInit 
	OR Errors.RH_BoMoldAIsMovingToMoldANotInPos OR Errors.RH_BoMoldAIsMovingTrMoldNotInPos OR Errors.RH_BoMoldBIsMovingToMoldBNotInPos OR Errors.RH_BoMoldBIsMovingTrMoldNotInPos
	OR Errors.RH_TaOutHorAIsMovingVertIsNotDown OR Errors.RH_TaOutHorBIsMovingVertIsNotDown OR Errors.RH_ToMoldAIsMovingBoMoldANotInPos OR Errors.RH_ToMoldBIsMovingBoMoldBNotInPos
	OR Errors.RH_TrMoldIsMovingBoMoldANotInPos OR Errors.RH_TrMoldIsMovingBoMoldBNotInPos OR Errors.RH_TrMoldIsMovingSprayBNotInPos OR Errors.RH_BotMoldAToCoolForTrMDown 
	OR Errors.RH_BotMoldBToCoolForTrMDown OR Errors.TempDeviationToHighA[1] OR Errors.TempDeviationToHighA[2] OR Errors.TempDeviationToHighA[3] OR Errors.TempDeviationToHighA[4]
	OR Errors.TempDeviationToHighA[5] OR Errors.TempDeviationToHighA[6] OR Errors.TempDeviationToHighB[1] OR Errors.TempDeviationToHighB[2] OR Errors.TempDeviationToHighB[3]
	OR Errors.TempDeviationToHighB[4] OR Errors.TempDeviationToHighB[5] OR Errors.TempDeviationToHighB[6];
END_ACTION

ACTION ErrorsTemperature:
(*Red hot safety regarding heating, block movement when top temperature deviates to much from bottom temperature*)
	SR_TempDeviationToHighA[1](SET1:=mxAutoMode AND
((BottomMoldA.HeatingZone[1].FB_Temperature.EngTempOut > TopMoldA.HeatingZone[1].FB_Temperature.EngTempOut + 40.0)  OR 
( BottomMoldA.HeatingZone[1].FB_Temperature.EngTempOut < TopMoldA.HeatingZone[1].FB_Temperature.EngTempOut - 40.0)), RESET:=mxReset, Q1=>Errors.TempDeviationToHighA[1]);

	SR_TempDeviationToHighA[2](SET1:=mxAutoMode AND
((BottomMoldA.HeatingZone[2].FB_Temperature.EngTempOut > TopMoldA.HeatingZone[2].FB_Temperature.EngTempOut + 40.0)  OR 
( BottomMoldA.HeatingZone[2].FB_Temperature.EngTempOut < TopMoldA.HeatingZone[2].FB_Temperature.EngTempOut - 40.0)), RESET:=mxReset, Q1=>Errors.TempDeviationToHighA[2]);

	SR_TempDeviationToHighA[3](SET1:=mxAutoMode AND
((BottomMoldA.HeatingZone[3].FB_Temperature.EngTempOut > TopMoldA.HeatingZone[3].FB_Temperature.EngTempOut + 40.0)  OR 
( BottomMoldA.HeatingZone[3].FB_Temperature.EngTempOut < TopMoldA.HeatingZone[3].FB_Temperature.EngTempOut - 40.0)), RESET:=mxReset, Q1=>Errors.TempDeviationToHighA[3]);

	SR_TempDeviationToHighA[4](SET1:=mxAutoMode AND
((BottomMoldA.HeatingZone[4].FB_Temperature.EngTempOut > TopMoldA.HeatingZone[4].FB_Temperature.EngTempOut + 40.0)  OR 
( BottomMoldA.HeatingZone[4].FB_Temperature.EngTempOut < TopMoldA.HeatingZone[4].FB_Temperature.EngTempOut - 40.0)), RESET:=mxReset, Q1=>Errors.TempDeviationToHighA[4]);

	SR_TempDeviationToHighA[5](SET1:=mxAutoMode AND
((BottomMoldA.HeatingZone[5].FB_Temperature.EngTempOut > TopMoldA.HeatingZone[5].FB_Temperature.EngTempOut + 40.0)  OR 
( BottomMoldA.HeatingZone[5].FB_Temperature.EngTempOut < TopMoldA.HeatingZone[5].FB_Temperature.EngTempOut - 40.0)), RESET:=mxReset, Q1=>Errors.TempDeviationToHighA[5]);

	SR_TempDeviationToHighA[6](SET1:=mxAutoMode AND
((BottomMoldA.HeatingZone[6].FB_Temperature.EngTempOut > TopMoldA.HeatingZone[6].FB_Temperature.EngTempOut + 40.0)  OR 
( BottomMoldA.HeatingZone[6].FB_Temperature.EngTempOut < TopMoldA.HeatingZone[6].FB_Temperature.EngTempOut - 40.0)), RESET:=mxReset, Q1=>Errors.TempDeviationToHighA[6]);



(*Red hot safety regarding heating, block movement when top temperature deviates to much from bottom temperature*)
	SR_TempDeviationToHighB[1](SET1:=mxAutoMode AND
((BottomMoldB.HeatingZone[1].FB_Temperature.EngTempOut > TopMoldB.HeatingZone[1].FB_Temperature.EngTempOut + 40.0)  OR 
( BottomMoldB.HeatingZone[1].FB_Temperature.EngTempOut < TopMoldB.HeatingZone[1].FB_Temperature.EngTempOut - 40.0)), RESET:=mxReset, Q1=>Errors.TempDeviationToHighB[1]);

	SR_TempDeviationToHighB[2](SET1:=mxAutoMode AND
((BottomMoldB.HeatingZone[2].FB_Temperature.EngTempOut > TopMoldB.HeatingZone[2].FB_Temperature.EngTempOut + 40.0)  OR 
( BottomMoldB.HeatingZone[2].FB_Temperature.EngTempOut < TopMoldB.HeatingZone[2].FB_Temperature.EngTempOut - 40.0)), RESET:=mxReset, Q1=>Errors.TempDeviationToHighB[2]);

	SR_TempDeviationToHighB[3](SET1:=mxAutoMode AND
((BottomMoldB.HeatingZone[3].FB_Temperature.EngTempOut > TopMoldB.HeatingZone[3].FB_Temperature.EngTempOut + 40.0)  OR 
( BottomMoldB.HeatingZone[3].FB_Temperature.EngTempOut < TopMoldB.HeatingZone[3].FB_Temperature.EngTempOut - 40.0)), RESET:=mxReset, Q1=>Errors.TempDeviationToHighB[3]);

	SR_TempDeviationToHighB[4](SET1:=mxAutoMode AND
((BottomMoldB.HeatingZone[4].FB_Temperature.EngTempOut > TopMoldB.HeatingZone[4].FB_Temperature.EngTempOut + 40.0)  OR 
( BottomMoldB.HeatingZone[4].FB_Temperature.EngTempOut < TopMoldB.HeatingZone[4].FB_Temperature.EngTempOut - 40.0)), RESET:=mxReset, Q1=>Errors.TempDeviationToHighB[4]);

